     // nicht verwendete Signale für den 1. Schritt und eventuell weitere Schritte
     (*#sxSendBuf.sxSTW1.Jog1          := False;
             #sxSendBuf.sxSTW1.Jog2          := False;
             #sxSendBuf.sxEPosSTW1.MdiTyp    := False;
             #sxSendBuf.sxEPosSTW1.MdiPos    := False;
             #sxSendBuf.sxEPosSTW1.MdiNeg    := False;
             #sxSendBuf.sxEPosSTW1.MdiSetup  := False;
             #sxSendBuf.sxEPosSTW2.SetRefPt  := False;
             #sxSendBuf.sxEPosSTW2.JogInc    := False;
             #sxSendBuf.sxEPosSTW2.RefStDi   := False;
             #sxSendBuf.sxEPosSTW2.RefTyp    := False;
             #sxSendBuf.sxSTW1.RefStart      := False;
             #sxSendBuf.sxEPosSTW1.TrvBit0   := False;
             #sxSendBuf.sxEPosSTW1.TrvBit1   := False;
             #sxSendBuf.sxEPosSTW1.TrvBit2   := False;
             #sxSendBuf.sxEPosSTW1.TrvBit3   := False;
             #sxSendBuf.sxEPosSTW1.TrvBit4   := False;
             #sxSendBuf.sxEPosSTW1.TrvBit5   := False;
             #sxSendBuf.sxEPosSTW1.MdiStart  := False;*)
     #sxSendBuf.STW1.%X8 := False;
     #sxSendBuf.STW1.%X9 := False;
     #sxSendBuf.EPosSTW1.%X8 := False;
     #sxSendBuf.EPosSTW1.%X9 := False;
     #sxSendBuf.EPosSTW1.%X10 := False;
     #sxSendBuf.EPosSTW1.%X14 := False;
     #sxSendBuf.EPosSTW2.%X1 := False;
     #sxSendBuf.EPosSTW2.%X5 := False;
     #sxSendBuf.EPosSTW2.%X9 := False;
     #sxSendBuf.EPosSTW2.%X8 := False;
     #sxSendBuf.STW1.%X11 := False;
     #sxSendBuf.EPosSTW1.%X0 := False;
     #sxSendBuf.EPosSTW1.%X1 := False;
     #sxSendBuf.EPosSTW1.%X2 := False;
     #sxSendBuf.EPosSTW1.%X3 := False;
     #sxSendBuf.EPosSTW1.%X4 := False;
     #sxSendBuf.EPosSTW1.%X5 := False;
     #sxSendBuf.EPosSTW1.%X15 := False;

     // Bei der Auswahl der Verfahrsätze entspricht die Position der Verfahrensatznummer 
     // Verfahrsatznummer aus der Position ermitteln und in die einzelnen Bit's aufteilen
     // Es sind die Verfahrsatznummern 0 - 63 möglich
     IF (DINT_TO_INT(#Position) < 0) OR (DINT_TO_INT(#Position) > 63) THEN
       // Fehler, ungültiger Verfahrsatznummer
       #swStatus := 16#8204;
       #Error := True;
     ELSE
       // Fehler wieder zurücknehmen, wenn er mal ausgelöst wurde
       IF #swStatus = 16#8204 THEN
         #swStatus := 16#7002;
         #Error := False;
       END_IF;

       // Verfahrsatznummer Bit 0 ermitteln
       IF (DINT_TO_WORD(#Position) AND W#16#01) = W#16#01 THEN
         //#sxSendBuf.sxEPosSTW1.TrvBit0 := True;
         #sxSendBuf.EPosSTW1.%X0 := True;
       END_IF;

       // Verfahrsatznummer Bit 1 ermitteln
       IF (DINT_TO_WORD(#Position) AND W#16#02) = W#16#02 THEN
         //#sxSendBuf.sxEPosSTW1.TrvBit1 := True;
         #sxSendBuf.EPosSTW1.%X1 := True;
       END_IF;

       // Verfahrsatznummer Bit 2 ermitteln
       IF (DINT_TO_WORD(#Position) AND W#16#04) = W#16#04 THEN
         //#sxSendBuf.sxEPosSTW1.TrvBit2 := True;
         #sxSendBuf.EPosSTW1.%X2 := True;
       END_IF;

       // Verfahrsatznummer Bit 3 ermitteln
       IF (DINT_TO_WORD(#Position) AND W#16#08) = W#16#08 THEN
         //#sxSendBuf.sxEPosSTW1.TrvBit3 := True;
         #sxSendBuf.EPosSTW1.%X3 := True;
       END_IF;

       // Verfahrsatznummer Bit 4 ermitteln
       IF (DINT_TO_WORD(#Position) AND W#16#10) = W#16#10 THEN
         //#sxSendBuf.sxEPosSTW1.TrvBit4 := True;
         #sxSendBuf.EPosSTW1.%X4 := True;
       END_IF;

       // Verfahrsatznummer Bit 5 ermitteln
       IF (DINT_TO_WORD(#Position) AND W#16#20) = W#16#20 THEN
         //#sxSendBuf.sxEPosSTW1.TrvBit5 := True;
         #sxSendBuf.EPosSTW1.%X5 := True;
       END_IF;

       // Nach dem Einschalten des Antriebes, prüfen ob der Antrieb betriebsbereit, in Operation ohne Fehler und Warnung ist, 
       // dann die Betriebsart MDI / Sollwertvorgabe Start gesetzt werden
       IF #sbOff1 AND #sbReady AND #sbIOp AND NOT #sbFault THEN

         #sxSendBuf.STW1.%X6 := #sbExecute;

         // "Fliegendes Referentieren" aktivieren
         // "Fliegendes Referenzieren" erst nach Einschalten des Antriebes möglich
         IF #sbRefTyp THEN

           // Referenziertyp auf "Fliegendes Referenzieren" einstellen
           //#sxSendBuf.sxEPosSTW2.RefTyp := True;
           #sxSendBuf.EPosSTW2.%X8 := True;

           // Nach der Anwahl des Referenziertyps "Fliegendes Referenzieren", 
           // ein Zyklus später kann das Referenzieren gestartet
           IF (#siRefTypCyc = 0) THEN
             #siRefTypCyc := #siRefTypCyc + 1;
           ELSE
             // Referenzieren starten
             //#sxSendBuf.sxSTW1.RefStart := True;
             #sxSendBuf.STW1.%X11 := True;
           END_IF;
         END_IF;
       END_IF;
     END_IF;

     // Hauptbetriebsart "Tippen" (Jogging)
     // Betriebsart "Tippen positiv" oder "Tippen negativ" angewählt 
   ELSIF #siModePos = 7 AND #sbModePos THEN

     // Antrieb einschalten
     //#sxSendBuf.sxSTW1.Off1 := #sbOff1;
     #sxSendBuf.STW1.%X0 := #sbOff1;

     // nicht verwendete Signale für den 1. Schritt und eventuell weitere Schritte
     (*#sxSendBuf.sxEPosSTW1.MdiStart := False;
             #sxSendBuf.sxEPosSTW2.JogInc   := False;
             #sxSendBuf.sxSTW1.Jog1         := False;
             #sxSendBuf.sxSTW1.Jog2         := False;
             #sxSendBuf.sxEPosSTW2.RefTyp   := False;
             #sxSendBuf.sxSTW1.RefStart     := False;
             #sxSendBuf.sxEPosSTW2.SetRefPt  := False;*)

     #sxSendBuf.EPosSTW1.%X15 := False;
     #sxSendBuf.EPosSTW2.%X5 := False;
     #sxSendBuf.STW1.%X8 := False;
     #sxSendBuf.STW1.%X9 := False;
     #sxSendBuf.EPosSTW2.%X8 := False;
     #sxSendBuf.STW1.%X11 := False;
     #sxSendBuf.EPosSTW2.%X1 := False;

     // Nach dem Einschalten des Antriebes, prüfen ob der Antrieb betriebsbereit, in Operation ohne Fehler und Warnung ist, 
     // dann kann Tippen positiv oder negativ gesetzt werden
     IF #sbOff1 AND #sbReady AND #sbIOp AND NOT #sbFault THEN

       // Tippen positiv
       IF #Jog1 AND NOT #Jog2 THEN
         //#sxSendBuf.sxSTW1.Jog1 := True;
         #sxSendBuf.STW1.%X8 := True;
       END_IF;

       // Tippen negativ
       IF #Jog2 AND NOT #Jog1 THEN
         //#sxSendBuf.sxSTW1.Jog2 := True;
         #sxSendBuf.STW1.%X9 := True;
       END_IF;

       // "Fliegendes Referentieren" aktivieren
       // "Fliegendes Referenzieren" erst nach Einschalten des Antriebes möglich
       IF #sbRefTyp THEN

         // Referenziertyp auf "Fliegendes Referenzieren" einstellen
         //#sxSendBuf.sxEPosSTW2.RefTyp := #FlyRef;
         #sxSendBuf.EPosSTW2.%X8 := #FlyRef;

         // Nach der Anwahl des Referenziertyps "Fliegendes Referenzieren", 
         // ein Zyklus später kann das Referenzieren gestartet
         IF (#siRefTypCyc = 0) THEN
           #siRefTypCyc := #siRefTypCyc + 1;
         ELSE
           // Referenzieren starten
           //#sxSendBuf.sxSTW1.RefStart := True;
           #sxSendBuf.STW1.%X11 := True;
         END_IF;
       END_IF;
     END_IF;

     // Betriebsart "Tippen positiv / Tippen negativ inkrementell" 
   ELSIF #siModePos = 8 AND #sbModePos THEN

     // Antrieb einschalten
     //#sxSendBuf.sxSTW1.OFF1 := #sbOff1;
     #sxSendBuf.STW1.%X0 := #sbOff1;

     // nicht verwendete Signale für den 1. Schritt und eventuell weitere Schritte
     (*#sxSendBuf.sxEPosSTW1.MdiStart := False;
             #sxSendBuf.sxEPosSTW2.JogInc   := False;
             #sxSendBuf.sxSTW1.Jog1         := False;
             #sxSendBuf.sxSTW1.Jog2         := False;
             #sxSendBuf.sxSTW1.RefStart     := False;
             #sxSendBuf.sxEPosSTW2.RefTyp   := False;
             #sxSendBuf.sxEPosSTW2.SetRefPt  := False;*)

     #sxSendBuf.EPosSTW1.%X15 := False;
     #sxSendBuf.EPosSTW2.%X5 := False;
     #sxSendBuf.STW1.%X8 := False;
     #sxSendBuf.STW1.%X9 := False;
     #sxSendBuf.STW1.%X11 := False;
     #sxSendBuf.EPosSTW2.%X8 := False;
     #sxSendBuf.EPosSTW2.%X1 := False;

     // Nach dem Einschalten des Antriebes, ein Paar Zyklen warten bevor Tippen negativ gesetzt werden kann
     // Nach dem Einschalten des Antriebes, prüfen ob der Antrieb betriebsbereit, in Operation ohne Fehler und Warnung ist, 
     // dann kann Tippen positiv oder negativ gesetzt werden
     IF #sbOff1 AND #sbReady AND #sbIOp AND NOT #sbFault THEN

       // Tippen inkrementell einstellen
       //#sxSendBuf.sxEPosSTW2.JogInc := True;
       #sxSendBuf.EPosSTW2.%X5 := True;

       #sbJogInc := True;

       // Nach dem Einstellen des Antriebes, ein Paar Zyklen warten bevor Tippen negativ oder Tippen positiv gesetz werden kann
       IF #sbJogInc AND (#siJogIncCyc = 0) THEN
         #siJogIncCyc := #siJogIncCyc + 1;
       ELSE

         // Tippen positiv oder negativ inkrementell zulassen
         IF #Jog1 XOR #Jog2 THEN

           //#sxSendBuf.sxSTW1.Jog1 := #Jog1;
           //#sxSendBuf.sxSTW1.Jog2 := #Jog2;
           #sxSendBuf.STW1.%X8 := #Jog1;
           #sxSendBuf.STW1.%X9 := #Jog2;
         END_IF;
       END_IF;

       // "Fliegendes Referentieren" aktivieren
       // "Fliegendes Referenzieren" erst nach Einschalten des Antriebes möglich
       IF #sbRefTyp THEN

         // Referenziertyp auf "Fliegendes Referenzieren" einstellen
         //#sxSendBuf.sxEPosSTW2.RefTyp := True;
         #sxSendBuf.EPosSTW2.%X8 := True;

         // Nach der Anwahl des Referenziertyps "Fliegendes Referenzieren", 
         // ein Zyklus später kann das Referenzieren gestartet
         IF (#siRefTypCyc = 0) THEN
           #siRefTypCyc := #siRefTypCyc + 1;
         ELSE
           // Referenzieren starten
           //#sxSendBuf.sxSTW1.RefStart := True;
           #sxSendBuf.STW1.%X11 := True;
         END_IF;
       END_IF;
     END_IF;
   ELSE
     // Werte wieder zurücknehmen
     (*#sxSendBuf.sxSTW1.Off1          := #Off1;
             #sxSendBuf.sxSTW1.RejTrvTsk     := False;
             #sxSendBuf.sxSTW1.TrvStart      := False;
             #sxSendBuf.sxEPosSTW1.MdiStart  := False;
             #sxSendBuf.sxSTW1.Jog1          := False;
             #sxSendBuf.sxSTW1.Jog2          := False;
             #sxSendBuf.sxEPosSTW1.MdiTyp    := False;
             #sxSendBuf.sxEPosSTW1.MdiPos    := False;
             #sxSendBuf.sxEPosSTW1.MdiNeg    := False;
             #sxSendBuf.sxEPosSTW1.MdiTrTyp  := False;
             #sxSendBuf.sxEPosSTW1.MdiSetup  := False;
             #sxSendBuf.sxEPosSTW2.SetRefPt  := False;
             #sxSendBuf.sxEPosSTW2.RefTyp    := False;
             #sxSendBuf.sxEPosSTW2.RefStDi   := False;
             #sxSendBuf.sxEPosSTW2.JogInc    := False;
             #sxSendBuf.sxSTW1.RefStart      := False;*)

     #sxSendBuf.STW1.%X0 := #EnableAxis;
     #sxSendBuf.STW1.%X4 := False;
     #sxSendBuf.STW1.%X6 := False;
     #sxSendBuf.EPosSTW1.%X15 := False;
     #sxSendBuf.STW1.%X8 := False;
     #sxSendBuf.STW1.%X9 := False;
     #sxSendBuf.EPosSTW1.%X8 := False;
     #sxSendBuf.EPosSTW1.%X9 := False;
     #sxSendBuf.EPosSTW1.%X10 := False;
     #sxSendBuf.EPosSTW1.%X12 := False;
     #sxSendBuf.EPosSTW1.%X14 := False;
     #sxSendBuf.EPosSTW2.%X1 := False;
     #sxSendBuf.EPosSTW2.%X8 := False;
     #sxSendBuf.EPosSTW2.%X9 := False;
     #sxSendBuf.EPosSTW2.%X5 := False;
     #sxSendBuf.STW1.%X11 := False;
   END_IF; // Hauptbetriebsart "Verfahrsätze" (Traversing Blocks)

   //Den Eingang ConfigEPos auf die einzelnen Bits im Telegramm verschalten
   #sxSendBuf.STW1.%X1 := #ConfigEPos.%X0;
   #sxSendBuf.STW1.%X2 := #ConfigEPos.%X1;
   #sxSendBuf.EPosSTW2.%X14 := #ConfigEPos.%X2;
   #sxSendBuf.EPosSTW2.%X15 := #ConfigEPos.%X3;
   #sxSendBuf.EPosSTW2.%X11 := #ConfigEPos.%X4;
   #sxSendBuf.EPosSTW2.%X10 := #ConfigEPos.%X5;
   #sxSendBuf.EPosSTW2.%X2 := #ConfigEPos.%X6;
   #sxSendBuf.STW1.%X13 := #ConfigEPos.%X7;
   #sxSendBuf.EPosSTW1.%X12 := #ConfigEPos.%X8;
   #sxSendBuf.STW2.%X0 := #ConfigEPos.%X9;
   #sxSendBuf.STW2.%X1 := #ConfigEPos.%X10;
   #sxSendBuf.STW2.%X2 := #ConfigEPos.%X11;
   #sxSendBuf.STW2.%X3 := #ConfigEPos.%X12;
   #sxSendBuf.STW2.%X4 := #ConfigEPos.%X13;
   #sxSendBuf.STW2.%X7 := #ConfigEPos.%X14;
   #sxSendBuf.STW1.%X12 := #ConfigEPos.%X15;
   #sxSendBuf.STW1.%X14 := #ConfigEPos.%X16;
   #sxSendBuf.STW1.%X15 := #ConfigEPos.%X17;
   #sxSendBuf.EPosSTW1.%X6 := #ConfigEPos.%X18;
   #sxSendBuf.EPosSTW1.%X7 := #ConfigEPos.%X19;
   #sxSendBuf.EPosSTW1.%X11 := #ConfigEPos.%X20;
   #sxSendBuf.EPosSTW1.%X13 := #ConfigEPos.%X21;
   #sxSendBuf.EPosSTW2.%X3 := #ConfigEPos.%X22;
   #sxSendBuf.EPosSTW2.%X4 := #ConfigEPos.%X23;
   #sxSendBuf.EPosSTW2.%X6 := #ConfigEPos.%X24;
   #sxSendBuf.EPosSTW2.%X7 := #ConfigEPos.%X25;
   #sxSendBuf.EPosSTW2.%X12 := #ConfigEPos.%X26;
   #sxSendBuf.EPosSTW2.%X13 := #ConfigEPos.%X27;
   #sxSendBuf.STW2.%X5 := #ConfigEPos.%X28;
   #sxSendBuf.STW2.%X6 := #ConfigEPos.%X29;
   #sxSendBuf.STW2.%X8 := #ConfigEPos.%X30;
   #sxSendBuf.STW2.%X9 := #ConfigEPos.%X31;


   #swSendBuf[0] := #sxSendBuf.STW1;
   #swSendBuf[1] := #sxSendBuf.EPosSTW1;
   #swSendBuf[2] := #sxSendBuf.EPosSTW2;
   #swSendBuf[3] := #sxSendBuf.STW2;
   #swSendBuf[4] := #sxSendBuf.OverrideV;
   #swSendBuf[5] := #sxSendBuf.Position.%W1;
   #swSendBuf[6] := #sxSendBuf.Position.%W0;
   #swSendBuf[7] := #sxSendBuf.Velocity.%W1;
   #swSendBuf[8] := #sxSendBuf.Velocity.%W0;
   #swSendBuf[9] := #sxSendBuf.OverrideA;
   #swSendBuf[10] := #sxSendBuf.OverrideD;
   #swSendBuf[11] := #sxSendBuf.Reserve;

   //Prozessdaten zur Signalbaugruppe schreiben
   #piRetSFC := DPWR_DAT(LADDR := #HWIDSTW,
                         RECORD := #swSendBuf);

   // Fehler der Rückmeldung ausgeben
   #DiagID := INT_TO_WORD(#piRetSFC);

   //kein Fehler beim Schreiben
   IF #piRetSFC = 0 THEN

     // Fehler wieder zurück nehmen
     IF (#swStatus = 16#8601) THEN
       #swStatus := 16#7002;
       #Error := False;
     END_IF;

     //Prozessdaten von der Signalbaugruppe lesen
     #piRetSFC := DPRD_DAT(LADDR := #HWIDZSW,
                           RECORD => #swRecvBuf);

     // Fehlermeldung der Rückmeldung ausgeben
     #DiagID := INT_TO_WORD(#piRetSFC);

     //Fehler beim Lesen (Profibus-Kommunikation unterbrochen)
     IF #piRetSFC <> 0 THEN

       // Fehler
       #Error := TRUE;
       #swStatus := 16#8600;

       // Zustandsworte löschen
       #sxRecvBuf.ZSW1 := W#16#0;
       #sxRecvBuf.EPosZSW1 := W#16#0;
       #sxRecvBuf.EPosZSW2 := W#16#0;
       #sxRecvBuf.ZSW2 := W#16#0;
       #sxRecvBuf.NotUsed := W#16#00;
       #sxRecvBuf.Position := DW#16#00;
       #sxRecvBuf.Velocity := DW#16#00;
       #sxRecvBuf.ErrNr := W#16#00;
       #sxRecvBuf.WarnNr := W#16#00;
       #sxRecvBuf.Reserve := W#16#00;

       // Werte auslesen
     ELSE

       // Fehler wieder zurück nehmen
       IF (#swStatus = 16#8600) THEN
         #swStatus := 16#7002;
         #Error := False;
       END_IF;

       #sxRecvBuf.ZSW1 := #swRecvBuf[0];
       #sxRecvBuf.EPosZSW1 := #swRecvBuf[1];
       #sxRecvBuf.EPosZSW2 := #swRecvBuf[2];
       #sxRecvBuf.ZSW2 := #swRecvBuf[3];
       #sxRecvBuf.NotUsed := #swRecvBuf[4];
       #sxRecvBuf.Position.%W1 := #swRecvBuf[5];
       #sxRecvBuf.Position.%W0 := #swRecvBuf[6];
       #sxRecvBuf.Velocity.%W1 := #swRecvBuf[7];
       #sxRecvBuf.Velocity.%W0 := #swRecvBuf[8];
       #sxRecvBuf.ErrNr := #swRecvBuf[9];
       #sxRecvBuf.WarnNr := #swRecvBuf[10];
       #sxRecvBuf.Reserve := #swRecvBuf[11];

       // ZSW1 aufbereiten
       //#Busy := #sxRecvBuf.sxZSW1.IOp;
       #sbBusy := #sxRecvBuf.ZSW1.%X2;

       // Fehler auswerten
       IF #sxRecvBuf.ZSW1.%X3 THEN
         #swStatus := 16#8401;
         #Error := True;
       ELSIF #sxRecvBuf.ZSW1.%X6 THEN
         #swStatus := 16#8402;
         #Error := True;
       ELSE
         // Fehler wieder zurück nehmen
         IF (#swStatus = 16#8401) OR (#swStatus = 16#8402) THEN
           #swStatus := 16#7002;
           #Error := False;
         END_IF;
       END_IF;

       // EPOS_ZSW1            
       // EPOS-Wort-1 BIT 00 --> 1 = Active traversing block bit 0
       //IF #sxRecvBuf.sxEPosZSW1.ActTrvBit0 THEN
       IF #sxRecvBuf.EPosZSW1.%X0 THEN
         #swEPosZSW1 := #swEPosZSW1 OR W#16#01;
       ELSE
         #swEPosZSW1 := #swEPosZSW1 AND W#16#FFFE;
       END_IF;

       // EPOS-Wort-1 Bit 01 --> 1 = Active traversing block bit 1
       //IF #sxRecvBuf.sxEPosZSW1.ActTrvBit1 THEN
       IF #sxRecvBuf.EPosZSW1.%X1 THEN
         #swEPosZSW1 := #swEPosZSW1 OR W#16#02;
       ELSE
         #swEPosZSW1 := #swEPosZSW1 AND W#16#FFFD;
       END_IF;

       // EPOS-Wort-1 Bit 02 --> 1 = Active traversing block bit 2
       //IF #sxRecvBuf.sxEPosZSW1.ActTrvBit2 THEN
       IF #sxRecvBuf.EPosZSW1.%X2 THEN
         #swEPosZSW1 := #swEPosZSW1 OR W#16#04;
       ELSE
         #swEPosZSW1 := #swEPosZSW1 AND W#16#FFFB;
       END_IF;

       // EPOS-Wort-1 Bit 03 --> 1 = Active traversing block bit 3
       //IF #sxRecvBuf.sxEPosZSW1.ActTrvBit3 THEN
       IF #sxRecvBuf.EPosZSW1.%X3 THEN
         #swEPosZSW1 := #swEPosZSW1 OR W#16#08;
       ELSE
         #swEPosZSW1 := #swEPosZSW1 AND W#16#FFF7;
       END_IF;(*

   *)

       // EPOS-Wort-1 Bit 04 --> 1 = Active traversing block bit 4 
       //IF #sxRecvBuf.sxEPosZSW1.ActTrvBit4 THEN
       IF #sxRecvBuf.EPosZSW1.%X4 THEN
         #swEPosZSW1 := #swEPosZSW1 OR W#16#10;
       ELSE
         #swEPosZSW1 := #swEPosZSW1 AND W#16#FFEF;
       END_IF;

       // EPOS-Wort-1 Bit 05 --> 1 = Active traversing block bit 5
       //IF #sxRecvBuf.sxEPosZSW1.ActTrvBit5 THEN
       IF #sxRecvBuf.EPosZSW1.%X5 THEN
         #swEPosZSW1 := #swEPosZSW1 OR W#16#20;
       ELSE
         #swEPosZSW1 := #swEPosZSW1 AND W#16#FFDF;
       END_IF;

       // EPOS-Wort-1 Bit 08 --> 1 = STOP cam minus active
       //IF #sxRecvBuf.sxEPosZSW1.StpCamMinAct THEN
       IF #sxRecvBuf.EPosZSW1.%X8 THEN
         #swEPosZSW1 := #swEPosZSW1 OR W#16#100;
       ELSE
         #swEPosZSW1 := #swEPosZSW1 AND W#16#FEFF;
       END_IF;

       // EPOS-Wort-1 Bit 09 --> 1 = STOP cam plus active
       //IF #sxRecvBuf.sxEPosZSW1.StpCamPlsAct THEN
       IF #sxRecvBuf.EPosZSW1.%X9 THEN
         #swEPosZSW1 := #swEPosZSW1 OR W#16#200;
       ELSE
         #swEPosZSW1 := #swEPosZSW1 AND W#16#FDFF;
       END_IF;

       // EPOS-Wort-1 Bit 10 --> 1 = Jogging active
       //IF #sxRecvBuf.sxEPosZSW1.JogAct THEN
       IF #sxRecvBuf.EPosZSW1.%X10 THEN
         #swEPosZSW1 := #swEPosZSW1 OR W#16#400;
       ELSE
         #swEPosZSW1 := #swEPosZSW1 AND W#16#FBFF;
       END_IF;

       // EPOS-Wort-1 Bit 11 --> 1 = Reference point approach active
       //IF #sxRecvBuf.sxEPosZSW1.RefAct THEN
       IF #sxRecvBuf.EPosZSW1.%X11 THEN
         #swEPosZSW1 := #swEPosZSW1 OR W#16#800;
       ELSE
         #swEPosZSW1 := #swEPosZSW1 AND W#16#F7FF;
       END_IF;

       // Anstossen des fliegenden Referenzieren prüfen, wenn die Rückmeldung fehlt dann wiederholen
       //IF NOT #sxRecvBuf.sxEPosZSW1.FlyRefAct AND #sbRefTyp AND #sxSendBuf.sxSTW1.RefStart THEN
       IF NOT #sxRecvBuf.EPosZSW1.%X12 AND #sbRefTyp AND #sxSendBuf.STW1.%X11 THEN

         // Wiederholung anstossen 
         IF #siRefActRetry < #siRetryMax THEN
           #siRefActRetry := #siRefActRetry + 1;

           // Referenzieren starten wieder wegnehmen
           //#sxSendBuf.sxSTW1.RefStart := False;
           #sxSendBuf.STW1.%X11 := False;
         ELSE

           // Fehlermeldung
           #swStatus := 16#8403;
           #Error := True;
         END_IF;
       ELSE

         // Fehler wieder zurücknehmen, wenn er mal ausgelöst wurde
         IF #swStatus = 16#8403 THEN
           #swStatus := 16#7002;
           #Error := False;
         END_IF;
         // Zähler zurücksetzen bei Rückmeldung fliegendes Referenzieren jetzt aktiviert oder bei Abwahl der Funktion
         IF (#sxRecvBuf.EPosZSW1.%X12 AND #sbRefTyp AND #sxSendBuf.STW1.%X11) OR NOT #FlyRef THEN
           #siRefActRetry := 0;
         END_IF;
       END_IF;

       // EPOS-Wort-1 Bit 12 --> 1 = Flying referencing active
       //IF #sxRecvBuf.sxEPosZSW1.FlyRefAct THEN
       IF #sxRecvBuf.EPosZSW1.%X12 THEN
         #swEPosZSW1 := #swEPosZSW1 OR W#16#1000;
       ELSE
         #swEPosZSW1 := #swEPosZSW1 AND W#16#EFFF;
       END_IF;

       // EPOS-Wort-1 Bit 13 --> 1 = Traversing block active
       //IF #sxRecvBuf.sxEPosZSW1.TrvBlAct THEN
       IF #sxRecvBuf.EPosZSW1.%X13 THEN
         #swEPosZSW1 := #swEPosZSW1 OR W#16#2000;
       ELSE
         #swEPosZSW1 := #swEPosZSW1 AND W#16#DFFF;
       END_IF;

       // EPOS-Wort-1 Bit 14 --> 1 = MDI setup active
       //IF #sxRecvBuf.sxEPosZSW1.MdiStupAct THEN
       IF #sxRecvBuf.EPosZSW1.%X14 THEN
         #swEPosZSW1 := #swEPosZSW1 OR W#16#4000;
       ELSE
         #swEPosZSW1 := #swEPosZSW1 AND W#16#BFFF;
       END_IF;

       // EPOS-Wort-1 Bit 15 --> 1 = MDI positing active
       //IF #sxRecvBuf.sxEPosZSW1.MdiPosAct THEN
       IF #sxRecvBuf.EPosZSW1.%X15 THEN
         #swEPosZSW1 := #swEPosZSW1 OR W#16#8000;
       ELSE
         #swEPosZSW1 := #swEPosZSW1 AND W#16#7FFF;
       END_IF;

       // EPOS_ZSW2 
       // EPOS-Wort-2 Bit 00 --> 1 = Tracking mode active
       //IF #sxRecvBuf.sxEPosZSW2.TrkModeAct THEN
       IF #sxRecvBuf.EPosZSW2.%X0 THEN
         #swEPosZSW2 := #swEPosZSW2 OR W#16#01;
       ELSE
         #swEPosZSW2 := #swEPosZSW2 AND W#16#FFFE;
       END_IF;

       // EPOS-Wort-2 Bit 01 --> 1 = Velocity limit active
       //IF #sxRecvBuf.sxEPosZSW2.VeloLimAct THEN
       IF #sxRecvBuf.EPosZSW2.%X1 THEN
         #swEPosZSW2 := #swEPosZSW2 OR W#16#02;
       ELSE
         #swEPosZSW2 := #swEPosZSW2 AND W#16#FFFD;
       END_IF;

       // EPOS-Wort-2 Bit 02 --> 1 = Setpoint static
       //IF #sxRecvBuf.sxEPosZSW2.SetPStat THEN
       IF #sxRecvBuf.EPosZSW2.%X2 THEN
         #swEPosZSW2 := #swEPosZSW2 OR W#16#04;
       ELSE
         #swEPosZSW2 := #swEPosZSW2 AND W#16#FFFB;
       END_IF;

       // EPOS-Wort-2 Bit 03 --> 1 = Printmark outside outer window
       //IF #sxRecvBuf.sxEPosZSW2.PrnMrkOut THEN
       IF #sxRecvBuf.EPosZSW2.%X3 THEN
         #swEPosZSW2 := #swEPosZSW2 OR W#16#08;
       ELSE
         #swEPosZSW2 := #swEPosZSW2 AND W#16#FFF7;
       END_IF;

       // EPOS-Wort-2 Bit 04 --> 1 = Axis forwards
       //IF #sxRecvBuf.sxEPosZSW2.FWD THEN
       IF #sxRecvBuf.EPosZSW2.%X4 THEN
         #swEPosZSW2 := #swEPosZSW2 OR W#16#10;
       ELSE
         #swEPosZSW2 := #swEPosZSW2 AND W#16#FFEF;
       END_IF;

       // EPOS-Wort-2 Bit 05 --> 1 = Axis backwards
       //IF #sxRecvBuf.sxEPosZSW2.BWD THEN
       IF #sxRecvBuf.EPosZSW2.%X5 THEN
         #swEPosZSW2 := #swEPosZSW2 OR W#16#20;
       ELSE
         #swEPosZSW2 := #swEPosZSW2 AND W#16#FFDF;
       END_IF;

       // EPOS-Wort-2 Bit 06 --> 1 = Software limit switch minus active
       //IF #sxRecvBuf.sxEPosZSW2.SftSwMinAct THEN
       IF #sxRecvBuf.EPosZSW2.%X6 THEN
         #swEPosZSW2 := #swEPosZSW2 OR W#16#40;
       ELSE
         #swEPosZSW2 := #swEPosZSW2 AND W#16#FFBF;
       END_IF;

       // EPOS-Wort-2 Bit 07 --> 1 = Software limit switch plus active
       //IF #sxRecvBuf.sxEPosZSW2.SftSwPlsAct THEN
       IF #sxRecvBuf.EPosZSW2.%X7 THEN
         #swEPosZSW2 := #swEPosZSW2 OR W#16#80;
       ELSE
         #swEPosZSW2 := #swEPosZSW2 AND W#16#FF7F;
       END_IF;

       // EPOS-Wort-2 Bit 08 --> 1 = Position actual value <= cam position 1
       //IF #sxRecvBuf.sxEPosZSW2.PosSmCam1 THEN
       IF #sxRecvBuf.EPosZSW2.%X8 THEN
         #swEPosZSW2 := #swEPosZSW2 OR W#16#100;
       ELSE
         #swEPosZSW2 := #swEPosZSW2 AND W#16#FEFF;
       END_IF;

       // EPOS-Wort-2 Bit 09 --> 1 = Position actual value <= cam position 2
       //IF #sxRecvBuf.sxEPosZSW2.PosSmCam2 THEN
       IF #sxRecvBuf.EPosZSW2.%X9 THEN
         #swEPosZSW2 := #swEPosZSW2 OR W#16#200;
       ELSE
         #swEPosZSW2 := #swEPosZSW2 AND W#16#FDFF;
       END_IF;

       // EPOS-Wort-2 Bit 10 --> 1 = Direct output 1 via traversing block
       //IF #sxRecvBuf.sxEPosZSW2.TrvOut1 THEN
       IF #sxRecvBuf.EPosZSW2.%X10 THEN
         #swEPosZSW2 := #swEPosZSW2 OR W#16#400;
       ELSE
         #swEPosZSW2 := #swEPosZSW2 AND W#16#FBFF;
       END_IF;

       // EPOS-Wort-2 Bit 11 --> 1 = Direct output 2 via traversing block
       //IF #sxRecvBuf.sxEPosZSW2.TrvOut2 THEN
       IF #sxRecvBuf.EPosZSW2.%X11 THEN
         #swEPosZSW2 := #swEPosZSW2 OR W#16#800;
       ELSE
         #swEPosZSW2 := #swEPosZSW2 AND W#16#F7FF;
       END_IF;

       // EPOS-Wort-2 Bit 12 --> 1 = Fixed STOP reached
       //IF #sxRecvBuf.sxEPosZSW2.FxStpRd THEN
       IF #sxRecvBuf.EPosZSW2.%X12 THEN
         #swEPosZSW2 := #swEPosZSW2 OR W#16#1000;
       ELSE
         #swEPosZSW2 := #swEPosZSW2 AND W#16#EFFF;
       END_IF;

       // EPOS-Wort-2 Bit 13 --> 1 = Fixed STOP clamping torque reached
       //IF #sxRecvBuf.sxEPosZSW2.FxStpTrRd THEN
       IF #sxRecvBuf.EPosZSW2.%X13 THEN
         #swEPosZSW2 := #swEPosZSW2 OR W#16#2000;
       ELSE
         #swEPosZSW2 := #swEPosZSW2 AND W#16#DFFF;
       END_IF;

       // EPOS-Wort-2 Bit 14 --> 1 = Traversing fixed STOP active
       //IF #sxRecvBuf.sxEPosZSW2.TrvFxStpAct THEN
       IF #sxRecvBuf.EPosZSW2.%X14 THEN
         #swEPosZSW2 := #swEPosZSW2 OR W#16#4000;
       ELSE
         #swEPosZSW2 := #swEPosZSW2 AND W#16#BFFF;
       END_IF;

       // EPOS-Wort-2 Bit 15 --> 1 = Traversing command active
       //IF #sxRecvBuf.sxEPosZSW2.CmdAct THEN
       IF #sxRecvBuf.EPosZSW2.%X15 THEN
         #swEPosZSW2 := #swEPosZSW2 OR W#16#8000;
       ELSE
         #swEPosZSW2 := #swEPosZSW2 AND W#16#7FFF;
       END_IF;

       #sbReady := #sxRecvBuf.ZSW1.%X1;

       #AxisEnabled := #sxRecvBuf.ZSW1.%X2;
       #sbIOp := #sxRecvBuf.ZSW1.%X2;

       #AxisError := #sxRecvBuf.ZSW1.%X3;
       #sbFault := #sxRecvBuf.ZSW1.%X3;

       #AxisWarn := #sxRecvBuf.ZSW1.%X7;
       #sbAlarm := #sxRecvBuf.ZSW1.%X7;

       #AxisPosOk := #sxRecvBuf.ZSW1.%X10;
       #AxisRef := #sxRecvBuf.ZSW1.%X11;
       #AxisSpFixed := #sxRecvBuf.ZSW1.%X13;

       #sbAccel := #sxRecvBuf.ZSW1.%X14;
       #sbDecel := #sxRecvBuf.ZSW1.%X15;

       #ActVelocity := DWORD_TO_DINT(#sxRecvBuf.Velocity);
       #ActPosition := DWORD_TO_DINT(#sxRecvBuf.Position);
       #ActMode := #ModePos;
       #ActWarn := #sxRecvBuf.WarnNr;
       #ActFault := #sxRecvBuf.ErrNr;

       #Lockout := #sxRecvBuf.ZSW1.%X6;
     END_IF;
   ELSE

     // Fehler
     #Error := TRUE;
     #swStatus := 16#8601;

   END_IF;

   // Initialisierung von Ausg㭧en
   #Status := #swStatus;
   #EPosZSW1 := #swEPosZSW1;
   #EPosZSW2 := #swEPosZSW2;
END_FUNCTION_BLOCK

// folder: General

FUNCTION_BLOCK "InOut"   // FB1, LAD
{ S7_Optimized_Access := 'TRUE' }
VERSION : 0.1
   VAR
      BaseDrive_LAD_Instance : "BaseDrive_LAD";
      CiftEl_Instance : "CiftEl";
   END_VAR
   VAR_TEMP
      bHmiServoStopButton : Bool;
      bDriveEnable : Bool;
   END_VAR
BEGIN

REGION Network 1: Cift El
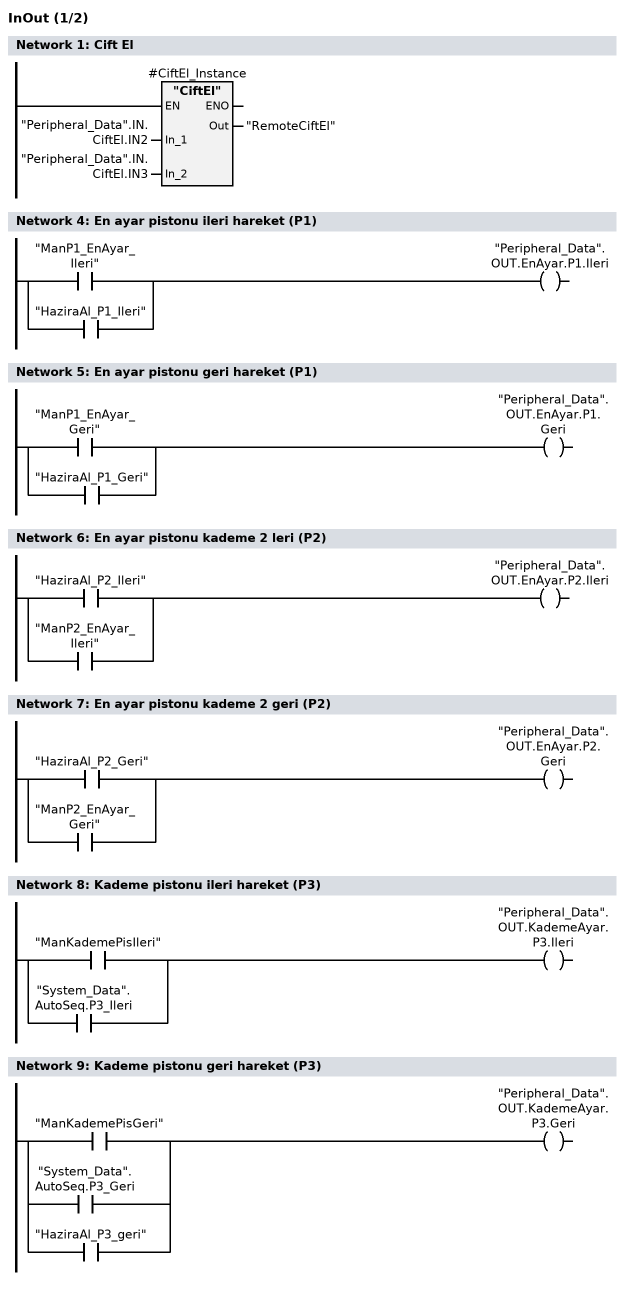
   RUNG wire#powerrail
      #CiftEl_Instance(In_1 := "Peripheral_Data".IN.CiftEl.IN2, In_2 := "Peripheral_Data".IN.CiftEl.IN3, Out => "RemoteCiftEl")
   END_RUNG
   // the same network as SCL:
   #CiftEl_Instance(In_1 := "Peripheral_Data".IN.CiftEl.IN2,   // "CiftEl"
                    In_2 := "Peripheral_Data".IN.CiftEl.IN3,
                    Out => "RemoteCiftEl");
END_REGION

REGION Network 2 (SCL): Servo veri yonetimi

   //********************************************//
   //******* Servo Poizsyona git işlemleri*******//
   "System_Data".CmdDrive.GoPos :=
   "ManServoGoPos" OR "System_Data".AutoSeq.GoPos
   OR "System_Data".AutoSeq.GoPos2 OR "HaziraAl_ServoGoPos"
   OR "ManServoGoHome" OR "ManServoGoPos2";

   //**********************************************//
   //********* Manuel jog kontrolleri*************//
   "System_Data".CmdDrive.Jog1 := "ManServoJog1";
   "System_Data".CmdDrive.Jog2 := "ManServoJog2";

   "System_Data".CmdDrive.SetReference := "System_Data".SystemMode.Man AND "HMI_Data".ServoButton.btnRefNokBelirle;
   "System_Data".CmdDrive.AckError := "System_Data".SystemMode.Man AND "HMI_Data".ServoButton.btnHataReset;
   //"System_Data".CmdDrive.Position := "Receipt".CurrentModel.Boy_C;

   //************************************************//
   //*********Servo hız bilgisi**********************//
   //

   "System_Data".CmdDrive.Velocity := 30.0;
   "System_Data".CmdDrive.Override := "HMI_Data".ServoData.txtJogOverride;  // jog hızı

   // IF "System_Data".SystemMode.Auto THEN
   //     //"System_Data".CmdDrive.Velocity := "HMI_Data".ServoData.txtVelocity;  //otomatik sekans hızı
   //     "System_Data".CmdDrive.Velocity := INT_TO_REAL("HMI_Data".ServoData.txtJogOverride);
   //     "System_Data".CmdDrive.Override := 100; 
   // ELSIF "System_Data".SystemMode.Man THEN
   //     "System_Data".CmdDrive.Velocity := INT_TO_REAL( "HMI_Data".ServoData.txtJogOverride );
   //     "System_Data".CmdDrive.Override := "HMI_Data".ServoData.txtJogOverride;  // jog hızı
   // END_IF;

   //***********************************************//
   //********** Home Konumu ************************//
   "System_Data".CmdDrive.HomePosition := 1560.0;
END_REGION

REGION Network 3 (SCL): Drive blogu
   // Hmi servo ekranı stop butonu sadece manuel modda çalışacak
   #bHmiServoStopButton := "HMI_Data".ServoButton.btnStop AND "System_Data".SystemMode.Man;
   #bDriveEnable := "System_Data".AutoSeq.StartedInfo
                   OR "HaziraAl_ServoGoPos"
                   OR "ManServoGoPos"
                   OR "ManServoGoPos2"
                   OR "ManServoGoHome"
                   OR "System_Data".CmdDrive.SetReference;

   #BaseDrive_LAD_Instance(Emergency := "Peripheral_Data".IN.Acil_Stop,
                           //Enable := #bDriveEnable,
                           Enable := "Peripheral_Data".IN.Acil_Stop AND NOT "HMI_Data".btnStop AND NOT #bHmiServoStopButton,
                           GoPos:="System_Data".CmdDrive.GoPos,
                           //GoHome:="System_Data".CmdDrive.GoHome,
                           SetReference:="System_Data".CmdDrive.SetReference,
                           Jog1:="System_Data".CmdDrive.Jog1,
                           Jog2:="System_Data".CmdDrive.Jog2,
                           Position:="System_Data".CmdDrive.Position,
                           Velocity:="System_Data".CmdDrive.Velocity,
                           Override:="System_Data".CmdDrive.Override,
                           AckError:="System_Data".CmdDrive.AckError,
                           HWDSTW:=280,
                           HWDZSW:=280,
                           Pos_Done=>"System_Data".CmdDrive.Pos_Done,
                           Busy=>"System_Data".CmdDrive.Busy,
                           Error=>"System_Data".CmdDrive.Error,
                           AxisError => "System_Data".CmdDrive.AxisError,
                           ErrorId=>"System_Data".CmdDrive.ErrorId,
                           ReferencedAxis=>"System_Data".CmdDrive.ReferencedAxis,
                           Message=>"System_Data".CmdDrive.Message,
                           ActPosition=>"System_Data".CmdDrive.ActPosition,
                           Alarm=>"System_Data".CmdDrive.Alarm,
                           //IsHomePosTol => "System_Data".CmdDrive.IsHomePosTol,
                           IsPosTol => "System_Data".CmdDrive.IsPosTol,
                           Standstill => "MemDrive_Standsill");

   "HMI_Data".ServoData.txtActPozisyon := "System_Data".CmdDrive.ActPosition;
END_REGION

REGION Network 4: En ayar pistonu ileri hareket (P1)
   RUNG wire#powerrail
      Contact( "ManP1_EnAyar_Ileri" )
      wire#w1
      Coil( "Peripheral_Data".OUT.EnAyar.P1.Ileri )
   END_RUNG
   RUNG wire#powerrail
      Contact( "HaziraAl_P1_Ileri" )
   END_RUNG wire#w1
   // the same network as SCL:
   "Peripheral_Data".OUT.EnAyar.P1.Ileri := "ManP1_EnAyar_Ileri" OR "HaziraAl_P1_Ileri";
END_REGION

REGION Network 5: En ayar pistonu geri hareket (P1)
   RUNG wire#powerrail
      Contact( "ManP1_EnAyar_Geri" )
      wire#w1
      Coil( "Peripheral_Data".OUT.EnAyar.P1.Geri )
   END_RUNG
   RUNG wire#powerrail
      Contact( "HaziraAl_P1_Geri" )
   END_RUNG wire#w1
   // the same network as SCL:
   "Peripheral_Data".OUT.EnAyar.P1.Geri := "ManP1_EnAyar_Geri" OR "HaziraAl_P1_Geri";
END_REGION

REGION Network 6: En ayar pistonu kademe 2 leri (P2)
   RUNG wire#powerrail
      Contact( "HaziraAl_P2_Ileri" )
      wire#w1
      Coil( "Peripheral_Data".OUT.EnAyar.P2.Ileri )
   END_RUNG
   RUNG wire#powerrail
      Contact( "ManP2_EnAyar_Ileri" )
   END_RUNG wire#w1
   // the same network as SCL:
   "Peripheral_Data".OUT.EnAyar.P2.Ileri := "HaziraAl_P2_Ileri" OR "ManP2_EnAyar_Ileri";
END_REGION

REGION Network 7: En ayar pistonu kademe 2 geri (P2)
   RUNG wire#powerrail
      Contact( "HaziraAl_P2_Geri" )
      wire#w1
      Coil( "Peripheral_Data".OUT.EnAyar.P2.Geri )
   END_RUNG
   RUNG wire#powerrail
      Contact( "ManP2_EnAyar_Geri" )
   END_RUNG wire#w1
   // the same network as SCL:
   "Peripheral_Data".OUT.EnAyar.P2.Geri := "HaziraAl_P2_Geri" OR "ManP2_EnAyar_Geri";
END_REGION

REGION Network 8: Kademe pistonu ileri hareket (P3)
   RUNG wire#powerrail
      Contact( "ManKademePisIleri" )
      wire#w1
      Coil( "Peripheral_Data".OUT.KademeAyar.P3.Ileri )
   END_RUNG
   RUNG wire#powerrail
      Contact( "System_Data".AutoSeq.P3_Ileri )
   END_RUNG wire#w1
   // the same network as SCL:
   "Peripheral_Data".OUT.KademeAyar.P3.Ileri := "ManKademePisIleri" OR "System_Data".AutoSeq.P3_Ileri;
END_REGION

REGION Network 9: Kademe pistonu geri hareket (P3)
   RUNG wire#powerrail
      Contact( "ManKademePisGeri" )
      wire#w1
      Coil( "Peripheral_Data".OUT.KademeAyar.P3.Geri )
   END_RUNG
   RUNG wire#powerrail
      Contact( "System_Data".AutoSeq.P3_Geri )
   END_RUNG wire#w1
   RUNG wire#powerrail
      Contact( "HaziraAl_P3_geri" )
   END_RUNG wire#w1
   // the same network as SCL:
   "Peripheral_Data".OUT.KademeAyar.P3.Geri := "ManKademePisGeri" OR "System_Data".AutoSeq.P3_Geri OR "HaziraAl_P3_geri";
END_REGION

REGION Network 10: Kenetleme pistonu ileri hareket (P4/P4B)
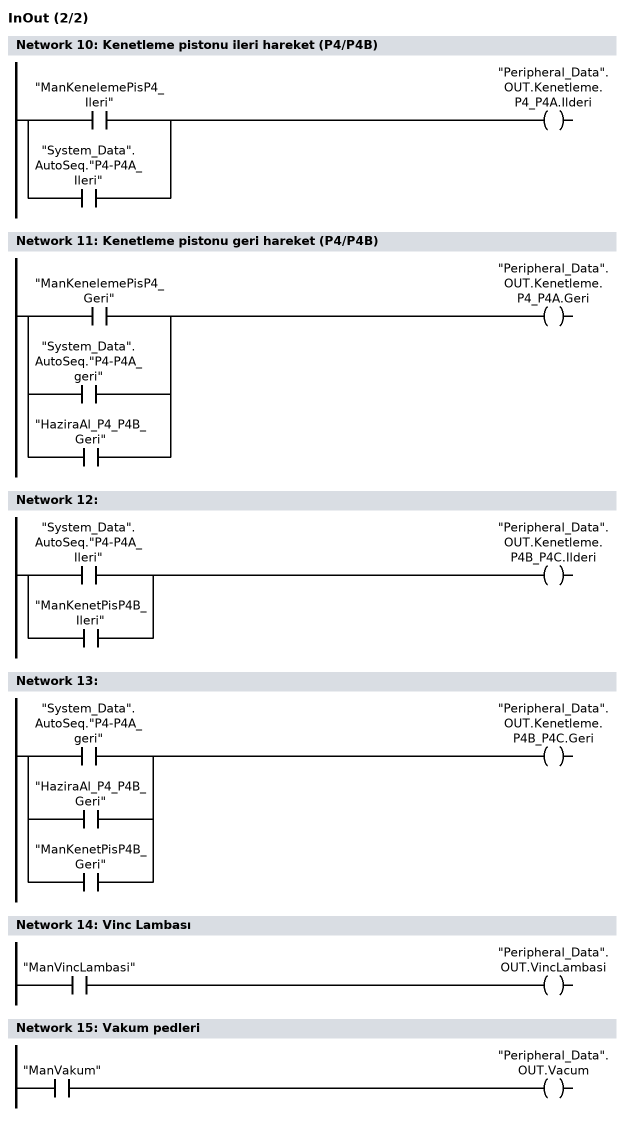
   RUNG wire#powerrail
      Contact( "ManKenelemePisP4_Ileri" )
      wire#w1
      Coil( "Peripheral_Data".OUT.Kenetleme.P4_P4A.Ilderi )
   END_RUNG
   RUNG wire#powerrail
      Contact( "System_Data".AutoSeq."P4-P4A_Ileri" )
   END_RUNG wire#w1
   // the same network as SCL:
   "Peripheral_Data".OUT.Kenetleme.P4_P4A.Ilderi := "ManKenelemePisP4_Ileri" OR "System_Data".AutoSeq."P4-P4A_Ileri";
END_REGION

REGION Network 11: Kenetleme pistonu geri hareket (P4/P4B)
   RUNG wire#powerrail
      Contact( "ManKenelemePisP4_Geri" )
      wire#w1
      Coil( "Peripheral_Data".OUT.Kenetleme.P4_P4A.Geri )
   END_RUNG
   RUNG wire#powerrail
      Contact( "System_Data".AutoSeq."P4-P4A_geri" )
   END_RUNG wire#w1
   RUNG wire#powerrail
      Contact( "HaziraAl_P4_P4B_Geri" )
   END_RUNG wire#w1
   // the same network as SCL:
   "Peripheral_Data".OUT.Kenetleme.P4_P4A.Geri := "ManKenelemePisP4_Geri" OR "System_Data".AutoSeq."P4-P4A_geri" OR "HaziraAl_P4_P4B_Geri";
END_REGION

REGION Network 12
   RUNG wire#powerrail
      Contact( "System_Data".AutoSeq."P4-P4A_Ileri" )
      wire#w1
      Coil( "Peripheral_Data".OUT.Kenetleme.P4B_P4C.Ilderi )
   END_RUNG
   RUNG wire#powerrail
      Contact( "ManKenetPisP4B_Ileri" )
   END_RUNG wire#w1
   // the same network as SCL:
   "Peripheral_Data".OUT.Kenetleme.P4B_P4C.Ilderi := "System_Data".AutoSeq."P4-P4A_Ileri" OR "ManKenetPisP4B_Ileri";
END_REGION

REGION Network 13
   RUNG wire#powerrail
      Contact( "System_Data".AutoSeq."P4-P4A_geri" )
      wire#w1
      Coil( "Peripheral_Data".OUT.Kenetleme.P4B_P4C.Geri )
   END_RUNG
   RUNG wire#powerrail
      Contact( "HaziraAl_P4_P4B_Geri" )
   END_RUNG wire#w1
   RUNG wire#powerrail
      Contact( "ManKenetPisP4B_Geri" )
   END_RUNG wire#w1
   // the same network as SCL:
   "Peripheral_Data".OUT.Kenetleme.P4B_P4C.Geri := "System_Data".AutoSeq."P4-P4A_geri" OR "HaziraAl_P4_P4B_Geri" OR "ManKenetPisP4B_Geri";
END_REGION

REGION Network 14: Vinc Lambası
   RUNG wire#powerrail
      Contact( "ManVincLambasi" )
      Coil( "Peripheral_Data".OUT.VincLambasi )
   END_RUNG
   // the same network as SCL:
   "Peripheral_Data".OUT.VincLambasi := "ManVincLambasi";
END_REGION

REGION Network 15: Vakum pedleri
   RUNG wire#powerrail
      Contact( "ManVakum" )
      Coil( "Peripheral_Data".OUT.Vacum )
   END_RUNG
   // the same network as SCL:
   "Peripheral_Data".OUT.Vacum := "ManVakum";
END_REGION
END_FUNCTION_BLOCK

FUNCTION "Peripheral" : Void   // FC2, SCL
{ S7_Optimized_Access := 'TRUE' }
VERSION : 0.1
BEGIN

   (**************************
   ******** INPUT *************
   **************************)

   "Peripheral_Data".IN.Acil_Stop := "I0.0";
   "Peripheral_Data".IN.CiftEl.IN1 := "I0.1";

   "Peripheral_Data".IN.CiftEl.IN2 := "I3.6";
   "Peripheral_Data".IN.CiftEl.IN3 := "I3.7";
   "Peripheral_Data".IN.VakumJen := "I0.2" OR "I0.3";

   "Peripheral_Data".IN.EnAyar.P1.Ileride := "I0.4";
   "Peripheral_Data".IN.EnAyar.P1.Geride := "I0.5";
   "Peripheral_Data".IN.EnAyar.P1A.Ileride := "I0.6";
   "Peripheral_Data".IN.EnAyar.P1A.Geride := "I0.7";

   "Peripheral_Data".IN.EnAyar.P2.Ileride := "I1.0";
   "Peripheral_Data".IN.EnAyar.P2.Geride := "I1.1";
   "Peripheral_Data".IN.EnAyar.P2A.Ileride := "I1.2";
   "Peripheral_Data".IN.EnAyar.P2A.Geride := "I1.3";

   "Peripheral_Data".IN.KademeAyar.P3.Ileride := "I1.4";
   "Peripheral_Data".IN.KademeAyar.P3.Geride := "I1.5";

   "Peripheral_Data".IN.Kenetleme.P4.Ilderide := "I2.0";
   "Peripheral_Data".IN.Kenetleme.P4.Geride := "I2.1";
   "Peripheral_Data".IN.Kenetleme.P4B.Ilderide := "I2.2";
   "Peripheral_Data".IN.Kenetleme.P4B.Geride := "I2.3";

   "Peripheral_Data".IN.VincUstuLamba := "I2.4";
   "Peripheral_Data".IN.ServoHomeSen := "I2.5";

   // "Peripheral_Data".IN.KademeAyar.P3A.Ileride := "I2.0";
   // "Peripheral_Data".IN.KademeAyar.P3A.Geride := "I2.1";

   // "Peripheral_Data".IN.Kenetleme.P4.Ilderide := "I2.2";
   // "Peripheral_Data".IN.Kenetleme.P4.Geride := "I2.3";
   // "Peripheral_Data".IN.Kenetleme.P4A.Ilderide := "I2.4";
   // "Peripheral_Data".IN.Kenetleme.P4A.Geride := "I2.5";

   // "Peripheral_Data".IN.Kenetleme.P4B.Ilderide := "I2.6";
   // "Peripheral_Data".IN.Kenetleme.P4B.Geride := "I2.7";
   // "Peripheral_Data".IN.Kenetleme.P4C.Ilderide := "I3.0";
   // "Peripheral_Data".IN.Kenetleme.P4C.Geride := "I3.1";

   // "Peripheral_Data".IN.VincUstuLamba := "I3.2";

   (**************************
   ******** OUTPUT ***********
   **************************)
   "Q0.0" := "Peripheral_Data".OUT.LAMBA.Kirmizi;
   "Q0.1" := "Peripheral_Data".OUT.LAMBA.Sari;
   "Q0.2" := "Peripheral_Data".OUT.LAMBA.Yesil;

   "Q0.3" := "Peripheral_Data".OUT.Vacum;
   "Q0.4" := "Peripheral_Data".OUT.VincLambasi;
   "Q0.5" := "Peripheral_Data".OUT.LAMBA.Buzzer;


   //*****************************************//
   //************* FESTO PROFINET ************//
   "Q4.0" := "Peripheral_Data".OUT.Kenetleme.P4B_P4C.Geri;
   "Q4.1" := "Peripheral_Data".OUT.Kenetleme.P4B_P4C.Ilderi;
   "Q4.2" := "Peripheral_Data".OUT.Kenetleme.P4_P4A.Geri;
   "Q4.3" := "Peripheral_Data".OUT.Kenetleme.P4_P4A.Ilderi;
   "Q4.4" := "Peripheral_Data".OUT.EnAyar.P1.Geri;
   "Q4.5" := "Peripheral_Data".OUT.EnAyar.P1.Ileri;
   "Q4.6" := "Peripheral_Data".OUT.EnAyar.P2.Geri;
   "Q4.7" := "Peripheral_Data".OUT.EnAyar.P2.Ileri;

   "Q5.0" := "Peripheral_Data".OUT.KademeAyar.P3.Geri;
   "Q5.1" := "Peripheral_Data".OUT.KademeAyar.P3.Ileri;
END_FUNCTION

FUNCTION "Station" : Void   // FC3, LAD
{ S7_Optimized_Access := 'TRUE' }
VERSION : 0.1
BEGIN

REGION Network 1: otomatik moda gecis
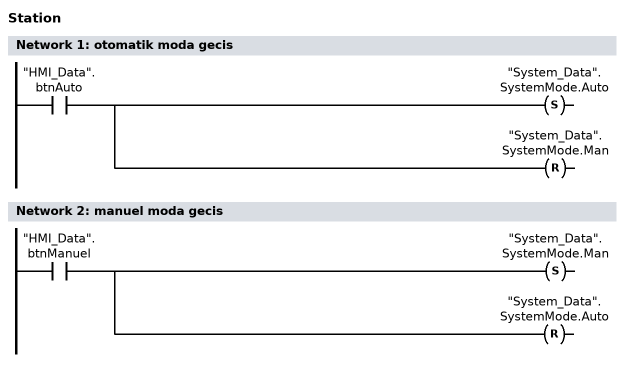
   RUNG wire#powerrail
      Contact( "HMI_Data".btnAuto )
      wire#w1
      S_Coil( "System_Data".SystemMode.Auto )
   END_RUNG
   RUNG wire#w1
      R_Coil( "System_Data".SystemMode.Man )
   END_RUNG
   // the same network as SCL:
   IF "HMI_Data".btnAuto THEN
       "System_Data".SystemMode.Auto := TRUE;
       "System_Data".SystemMode.Man := FALSE;
   END_IF;
END_REGION

REGION Network 2: manuel moda gecis
   RUNG wire#powerrail
      Contact( "HMI_Data".btnManuel )
      wire#w1
      S_Coil( "System_Data".SystemMode.Man )
   END_RUNG
   RUNG wire#w1
      R_Coil( "System_Data".SystemMode.Auto )
   END_RUNG
   // the same network as SCL:
   IF "HMI_Data".btnManuel THEN
       "System_Data".SystemMode.Man := TRUE;
       "System_Data".SystemMode.Auto := FALSE;
   END_IF;
END_REGION
END_FUNCTION

FUNCTION "HMI" : Void   // FC5, LAD
{ S7_Optimized_Access := 'TRUE' }
VERSION : 0.1
BEGIN

REGION Network 2 (SCL)
   // en ayar psitonu izleme 
   "HMI_Data".Status.EnAyarPis.P1.Ileride := "Peripheral_Data".IN.EnAyar.P1.Ileride
   AND "Peripheral_Data".IN.EnAyar.P1A.Ileride;
   "HMI_Data".Status.EnAyarPis.P2.Ileride := "Peripheral_Data".IN.EnAyar.P2.Ileride
   AND "Peripheral_Data".IN.EnAyar.P2A.Ileride;

   "HMI_Data".Status.EnAyarPis.P1.Geride := "Peripheral_Data".IN.EnAyar.P1.Geride
   AND "Peripheral_Data".IN.EnAyar.P1A.Geride;
   "HMI_Data".Status.EnAyarPis.P2.Geride := "Peripheral_Data".IN.EnAyar.P2.Geride
   AND "Peripheral_Data".IN.EnAyar.P2A.Geride;

   // kademe psitonu izleme 
   "HMI_Data".Status.KademePis_P3.Ileride := "Peripheral_Data".IN.KademeAyar.P3.Ileride;

   "HMI_Data".Status.KademePis_P3.Geride := "Peripheral_Data".IN.KademeAyar.P3.Geride;

   // kenetleme psitonu izleme
   "HMI_Data".Status.KenetlemePis_P4.Ileride := "Peripheral_Data".IN.Kenetleme.P4.Ilderide
   AND "Peripheral_Data".IN.Kenetleme.P4B.Ilderide;

   "HMI_Data".Status.KenetlemePis_P4.Geride := "Peripheral_Data".IN.Kenetleme.P4.Geride
   AND "Peripheral_Data".IN.Kenetleme.P4B.Geride;

   //Sistem secilen modele gore konumu hazir ise hazira al butonu yeşil olsun
   IF "Receipt".CurrentModel.Class = 0 THEN
       "System_Data".Ready := "ClassA_Hazir";
   ELSIF "Receipt".CurrentModel.Class = 1 THEN
       "System_Data".Ready := "ClassE_Hazir";
   ELSIF "Receipt".CurrentModel.Class = 2 THEN
       "System_Data".Ready := "ClassF_Hazir";
   ELSE
       "System_Data".Ready := false;
   END_IF;
END_REGION
END_FUNCTION

FUNCTION "UyariLambasi" : Void   // FC6, LAD
{ S7_Optimized_Access := 'TRUE' }
VERSION : 0.1
   VAR_TEMP
      wCheckAlarmWord : Word;   // "03FF" - piston timeout ve servo arıza bilgileri
      bCheckAlarmWord : Bool;
   END_VAR
BEGIN

REGION Network 1: Yesil lamba
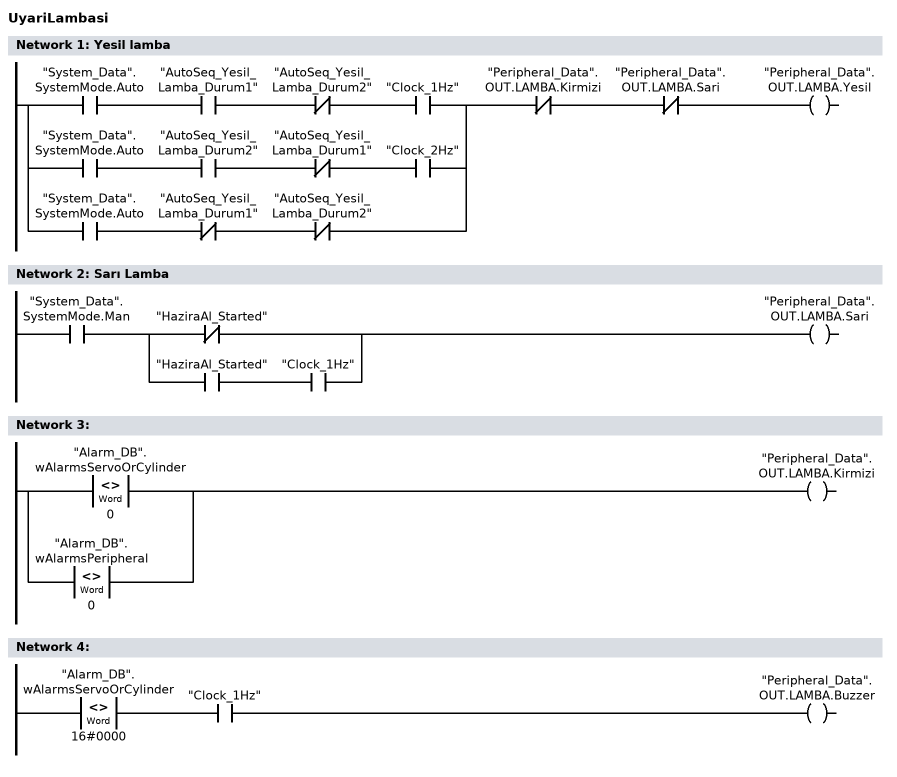
   RUNG wire#powerrail
      Contact( "System_Data".SystemMode.Auto )
      Contact( "AutoSeq_Yesil_Lamba_Durum1" )
      I_Contact( "AutoSeq_Yesil_Lamba_Durum2" )
      Contact( "Clock_1Hz" )
      wire#w1
      I_Contact( "Peripheral_Data".OUT.LAMBA.Kirmizi )
      I_Contact( "Peripheral_Data".OUT.LAMBA.Sari )
      Coil( "Peripheral_Data".OUT.LAMBA.Yesil )
   END_RUNG
   RUNG wire#powerrail
      Contact( "System_Data".SystemMode.Auto )
      Contact( "AutoSeq_Yesil_Lamba_Durum2" )
      I_Contact( "AutoSeq_Yesil_Lamba_Durum1" )
      Contact( "Clock_2Hz" )
   END_RUNG wire#w1
   RUNG wire#powerrail
      Contact( "System_Data".SystemMode.Auto )
      I_Contact( "AutoSeq_Yesil_Lamba_Durum1" )
      I_Contact( "AutoSeq_Yesil_Lamba_Durum2" )
   END_RUNG wire#w1
   // the same network as SCL:
   "Peripheral_Data".OUT.LAMBA.Yesil := (("System_Data".SystemMode.Auto AND "AutoSeq_Yesil_Lamba_Durum1" AND NOT "AutoSeq_Yesil_Lamba_Durum2" AND "Clock_1Hz") OR ("System_Data".SystemMode.Auto AND "AutoSeq_Yesil_Lamba_Durum2" AND NOT "AutoSeq_Yesil_Lamba_Durum1" AND "Clock_2Hz") OR ("System_Data".SystemMode.Auto AND NOT "AutoSeq_Yesil_Lamba_Durum1" AND NOT "AutoSeq_Yesil_Lamba_Durum2")) AND NOT "Peripheral_Data".OUT.LAMBA.Kirmizi AND NOT "Peripheral_Data".OUT.LAMBA.Sari;
END_REGION

REGION Network 2: Sarı Lamba
   RUNG wire#powerrail
      Contact( "System_Data".SystemMode.Man )
      wire#w1
      I_Contact( "HaziraAl_Started" )
      wire#w2
      Coil( "Peripheral_Data".OUT.LAMBA.Sari )
   END_RUNG
   RUNG wire#w1
      Contact( "HaziraAl_Started" )
      Contact( "Clock_1Hz" )
   END_RUNG wire#w2
   // the same network as SCL:
   "Peripheral_Data".OUT.LAMBA.Sari := "System_Data".SystemMode.Man AND (NOT "HaziraAl_Started" OR ("HaziraAl_Started" AND "Clock_1Hz"));
END_REGION

REGION Network 3
   RUNG wire#powerrail
      { S7_Templates := "SrcType := Word" } NE_Contact(in1 := "Alarm_DB".wAlarmsServoOrCylinder, in2 := 0)
      wire#w1
      Coil( "Peripheral_Data".OUT.LAMBA.Kirmizi )
   END_RUNG
   RUNG wire#powerrail
      { S7_Templates := "SrcType := Word" } NE_Contact(in1 := "Alarm_DB".wAlarmsPeripheral, in2 := 0)
   END_RUNG wire#w1
   // the same network as SCL:
   "Peripheral_Data".OUT.LAMBA.Kirmizi := ("Alarm_DB".wAlarmsServoOrCylinder <> 0) OR ("Alarm_DB".wAlarmsPeripheral <> 0);
END_REGION

REGION Network 4
   RUNG wire#powerrail
      { S7_Templates := "SrcType := Word" } NE_Contact(in1 := "Alarm_DB".wAlarmsServoOrCylinder, in2 := 16#0000)
      Contact( "Clock_1Hz" )
      Coil( "Peripheral_Data".OUT.LAMBA.Buzzer )
   END_RUNG
   // the same network as SCL:
   "Peripheral_Data".OUT.LAMBA.Buzzer := ("Alarm_DB".wAlarmsServoOrCylinder <> 16#0000) AND "Clock_1Hz";
END_REGION
END_FUNCTION

// folder: Manuel

FUNCTION_BLOCK "Manuel"   // FB3, LAD
{ S7_Optimized_Access := 'TRUE' }
VERSION : 0.1
   VAR_TEMP   // added for the SCL form of the ladder/FBD networks
      _w1 : Bool;
   END_VAR
BEGIN

REGION Network 1: Servo Manuel Jog 1
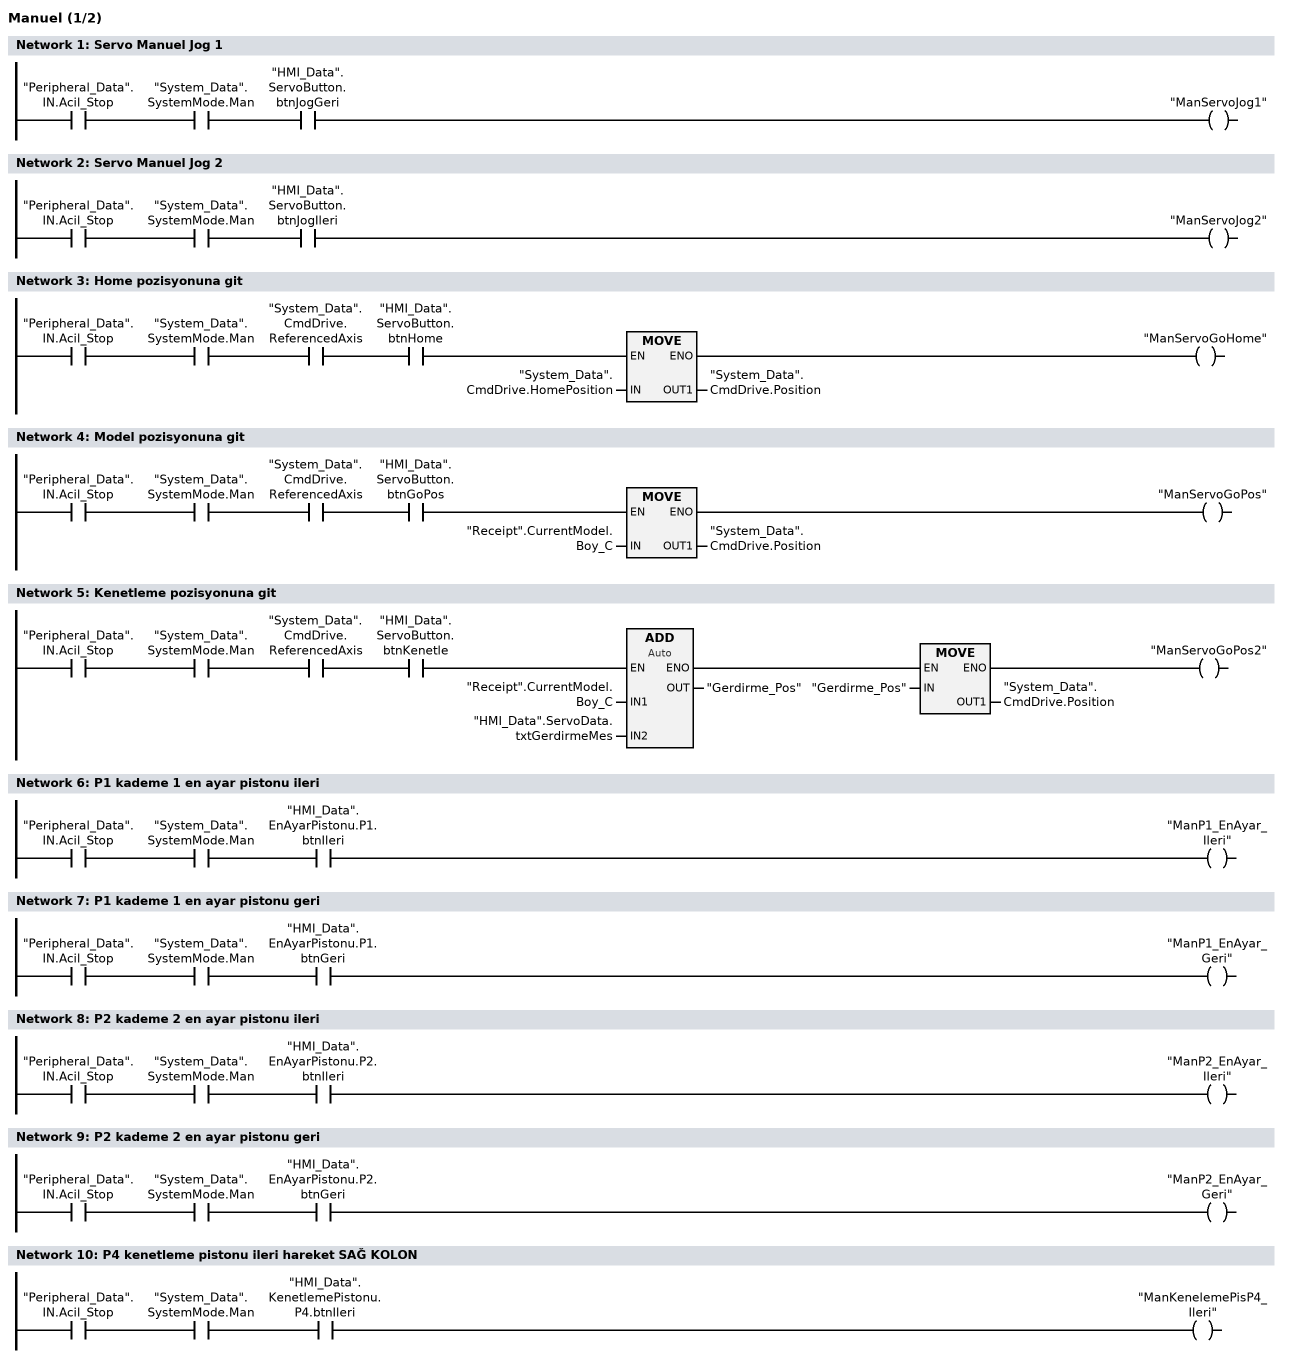
   RUNG wire#powerrail
      Contact( "Peripheral_Data".IN.Acil_Stop )
      Contact( "System_Data".SystemMode.Man )
      Contact( "HMI_Data".ServoButton.btnJogGeri )
      Coil( "ManServoJog1" )
   END_RUNG
   // the same network as SCL:
   "ManServoJog1" := "Peripheral_Data".IN.Acil_Stop AND "System_Data".SystemMode.Man AND "HMI_Data".ServoButton.btnJogGeri;
END_REGION

REGION Network 2: Servo Manuel Jog 2
   RUNG wire#powerrail
      Contact( "Peripheral_Data".IN.Acil_Stop )
      Contact( "System_Data".SystemMode.Man )
      Contact( "HMI_Data".ServoButton.btnJogIleri )
      Coil( "ManServoJog2" )
   END_RUNG
   // the same network as SCL:
   "ManServoJog2" := "Peripheral_Data".IN.Acil_Stop AND "System_Data".SystemMode.Man AND "HMI_Data".ServoButton.btnJogIleri;
END_REGION

REGION Network 3: Home pozisyonuna git
   RUNG wire#powerrail
      Contact( "Peripheral_Data".IN.Acil_Stop )
      Contact( "System_Data".SystemMode.Man )
      Contact( "System_Data".CmdDrive.ReferencedAxis )
      Contact( "HMI_Data".ServoButton.btnHome )
      Move(in := "System_Data".CmdDrive.HomePosition, out1 => "System_Data".CmdDrive.Position)
      Coil( "ManServoGoHome" )
   END_RUNG
   // the same network as SCL:
   #_w1 := "Peripheral_Data".IN.Acil_Stop AND "System_Data".SystemMode.Man AND "System_Data".CmdDrive.ReferencedAxis AND "HMI_Data".ServoButton.btnHome;
   IF #_w1 THEN "System_Data".CmdDrive.Position := "System_Data".CmdDrive.HomePosition; END_IF;
   "ManServoGoHome" := #_w1;
END_REGION

REGION Network 4: Model pozisyonuna git
   RUNG wire#powerrail
      Contact( "Peripheral_Data".IN.Acil_Stop )
      Contact( "System_Data".SystemMode.Man )
      Contact( "System_Data".CmdDrive.ReferencedAxis )
      Contact( "HMI_Data".ServoButton.btnGoPos )
      Move(in := "Receipt".CurrentModel.Boy_C, out1 => "System_Data".CmdDrive.Position)
      Coil( "ManServoGoPos" )
   END_RUNG
   // the same network as SCL:
   #_w1 := "Peripheral_Data".IN.Acil_Stop AND "System_Data".SystemMode.Man AND "System_Data".CmdDrive.ReferencedAxis AND "HMI_Data".ServoButton.btnGoPos;
   IF #_w1 THEN "System_Data".CmdDrive.Position := "Receipt".CurrentModel.Boy_C; END_IF;
   "ManServoGoPos" := #_w1;
END_REGION

REGION Network 5: Kenetleme pozisyonuna git
   RUNG wire#powerrail
      Contact( "Peripheral_Data".IN.Acil_Stop )
      Contact( "System_Data".SystemMode.Man )
      Contact( "System_Data".CmdDrive.ReferencedAxis )
      Contact( "HMI_Data".ServoButton.btnKenetle )
      Add(in1 := "Receipt".CurrentModel.Boy_C, in2 := "HMI_Data".ServoData.txtGerdirmeMes, out => "Gerdirme_Pos")
      Move(in := "Gerdirme_Pos", out1 => "System_Data".CmdDrive.Position)
      Coil( "ManServoGoPos2" )
   END_RUNG
   // the same network as SCL:
   #_w1 := "Peripheral_Data".IN.Acil_Stop AND "System_Data".SystemMode.Man AND "System_Data".CmdDrive.ReferencedAxis AND "HMI_Data".ServoButton.btnKenetle;
   IF #_w1 THEN
       "Gerdirme_Pos" := "Receipt".CurrentModel.Boy_C + "HMI_Data".ServoData.txtGerdirmeMes;
       "System_Data".CmdDrive.Position := "Gerdirme_Pos";
   END_IF;
   "ManServoGoPos2" := #_w1;
END_REGION

REGION Network 6: P1 kademe 1 en ayar pistonu ileri
   RUNG wire#powerrail
      Contact( "Peripheral_Data".IN.Acil_Stop )
      Contact( "System_Data".SystemMode.Man )
      Contact( "HMI_Data".EnAyarPistonu.P1.btnIleri )
      Coil( "ManP1_EnAyar_Ileri" )
   END_RUNG
   // the same network as SCL:
   "ManP1_EnAyar_Ileri" := "Peripheral_Data".IN.Acil_Stop AND "System_Data".SystemMode.Man AND "HMI_Data".EnAyarPistonu.P1.btnIleri;
END_REGION

REGION Network 7: P1 kademe 1 en ayar pistonu geri
   RUNG wire#powerrail
      Contact( "Peripheral_Data".IN.Acil_Stop )
      Contact( "System_Data".SystemMode.Man )
      Contact( "HMI_Data".EnAyarPistonu.P1.btnGeri )
      Coil( "ManP1_EnAyar_Geri" )
   END_RUNG
   // the same network as SCL:
   "ManP1_EnAyar_Geri" := "Peripheral_Data".IN.Acil_Stop AND "System_Data".SystemMode.Man AND "HMI_Data".EnAyarPistonu.P1.btnGeri;
END_REGION

REGION Network 8: P2 kademe 2 en ayar pistonu ileri
   RUNG wire#powerrail
      Contact( "Peripheral_Data".IN.Acil_Stop )
      Contact( "System_Data".SystemMode.Man )
      Contact( "HMI_Data".EnAyarPistonu.P2.btnIleri )
      Coil( "ManP2_EnAyar_Ileri" )
   END_RUNG
   // the same network as SCL:
   "ManP2_EnAyar_Ileri" := "Peripheral_Data".IN.Acil_Stop AND "System_Data".SystemMode.Man AND "HMI_Data".EnAyarPistonu.P2.btnIleri;
END_REGION

REGION Network 9: P2 kademe 2 en ayar pistonu geri
   RUNG wire#powerrail
      Contact( "Peripheral_Data".IN.Acil_Stop )
      Contact( "System_Data".SystemMode.Man )
      Contact( "HMI_Data".EnAyarPistonu.P2.btnGeri )
      Coil( "ManP2_EnAyar_Geri" )
   END_RUNG
   // the same network as SCL:
   "ManP2_EnAyar_Geri" := "Peripheral_Data".IN.Acil_Stop AND "System_Data".SystemMode.Man AND "HMI_Data".EnAyarPistonu.P2.btnGeri;
END_REGION

REGION Network 10: P4 kenetleme pistonu ileri hareket SAĞ KOLON
   RUNG wire#powerrail
      Contact( "Peripheral_Data".IN.Acil_Stop )
      Contact( "System_Data".SystemMode.Man )
      Contact( "HMI_Data".KenetlemePistonu.P4.btnIleri )
      Coil( "ManKenelemePisP4_Ileri" )
   END_RUNG
   // the same network as SCL:
   "ManKenelemePisP4_Ileri" := "Peripheral_Data".IN.Acil_Stop AND "System_Data".SystemMode.Man AND "HMI_Data".KenetlemePistonu.P4.btnIleri;
END_REGION

REGION Network 11: P4 kenetleme pistonu geri hareket (SAĞ KOLON)
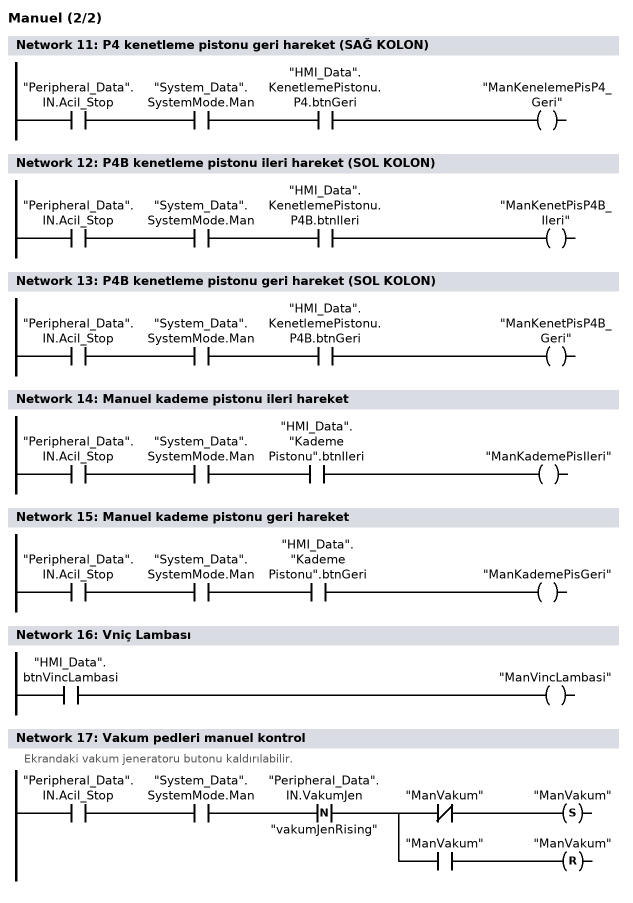
   RUNG wire#powerrail
      Contact( "Peripheral_Data".IN.Acil_Stop )
      Contact( "System_Data".SystemMode.Man )
      Contact( "HMI_Data".KenetlemePistonu.P4.btnGeri )
      Coil( "ManKenelemePisP4_Geri" )
   END_RUNG
   // the same network as SCL:
   "ManKenelemePisP4_Geri" := "Peripheral_Data".IN.Acil_Stop AND "System_Data".SystemMode.Man AND "HMI_Data".KenetlemePistonu.P4.btnGeri;
END_REGION

REGION Network 12: P4B kenetleme pistonu ileri hareket (SOL KOLON)
   RUNG wire#powerrail
      Contact( "Peripheral_Data".IN.Acil_Stop )
      Contact( "System_Data".SystemMode.Man )
      Contact( "HMI_Data".KenetlemePistonu.P4B.btnIleri )
      Coil( "ManKenetPisP4B_Ileri" )
   END_RUNG
   // the same network as SCL:
   "ManKenetPisP4B_Ileri" := "Peripheral_Data".IN.Acil_Stop AND "System_Data".SystemMode.Man AND "HMI_Data".KenetlemePistonu.P4B.btnIleri;
END_REGION

REGION Network 13: P4B kenetleme pistonu geri hareket (SOL KOLON)
   RUNG wire#powerrail
      Contact( "Peripheral_Data".IN.Acil_Stop )
      Contact( "System_Data".SystemMode.Man )
      Contact( "HMI_Data".KenetlemePistonu.P4B.btnGeri )
      Coil( "ManKenetPisP4B_Geri" )
   END_RUNG
   // the same network as SCL:
   "ManKenetPisP4B_Geri" := "Peripheral_Data".IN.Acil_Stop AND "System_Data".SystemMode.Man AND "HMI_Data".KenetlemePistonu.P4B.btnGeri;
END_REGION

REGION Network 14: Manuel kademe pistonu ileri hareket
   RUNG wire#powerrail
      Contact( "Peripheral_Data".IN.Acil_Stop )
      Contact( "System_Data".SystemMode.Man )
      Contact( "HMI_Data"."Kademe Pistonu".btnIleri )
      Coil( "ManKademePisIleri" )
   END_RUNG
   // the same network as SCL:
   "ManKademePisIleri" := "Peripheral_Data".IN.Acil_Stop AND "System_Data".SystemMode.Man AND "HMI_Data"."Kademe Pistonu".btnIleri;
END_REGION

REGION Network 15: Manuel kademe pistonu geri hareket
   RUNG wire#powerrail
      Contact( "Peripheral_Data".IN.Acil_Stop )
      Contact( "System_Data".SystemMode.Man )
      Contact( "HMI_Data"."Kademe Pistonu".btnGeri )
      Coil( "ManKademePisGeri" )
   END_RUNG
   // the same network as SCL:
   "ManKademePisGeri" := "Peripheral_Data".IN.Acil_Stop AND "System_Data".SystemMode.Man AND "HMI_Data"."Kademe Pistonu".btnGeri;
END_REGION

REGION Network 16: Vniç Lambası
   RUNG wire#powerrail
      Contact( "HMI_Data".btnVincLambasi )
      Coil( "ManVincLambasi" )
   END_RUNG
   // the same network as SCL:
   "ManVincLambasi" := "HMI_Data".btnVincLambasi;
END_REGION

REGION Network 17: Vakum pedleri manuel kontrol
   // Ekrandaki vakum jeneratoru butonu kaldırılabilir.
   RUNG wire#powerrail
      Contact( "Peripheral_Data".IN.Acil_Stop )
      Contact( "System_Data".SystemMode.Man )
      N_Contact(operand := "Peripheral_Data".IN.VakumJen, bit := "vakumJenRising")
      wire#w1
      I_Contact( "ManVakum" )
      S_Coil( "ManVakum" )
   END_RUNG
   RUNG wire#w1
      Contact( "ManVakum" )
      R_Coil( "ManVakum" )
   END_RUNG
   // the same network as SCL:
   #_w1 := "Peripheral_Data".IN.Acil_Stop AND "System_Data".SystemMode.Man AND NOT "Peripheral_Data".IN.VakumJen AND "vakumJenRising";   // falling edge of "Peripheral_Data".IN.VakumJen
   "vakumJenRising" := "Peripheral_Data".IN.VakumJen;
   IF #_w1 AND NOT "ManVakum" THEN "ManVakum" := TRUE; END_IF;
   IF #_w1 AND "ManVakum" THEN "ManVakum" := FALSE; END_IF;
END_REGION
END_FUNCTION_BLOCK

// folder: Otomatik

FUNCTION_BLOCK "Otomatik_Seq_LAD"   // FB5, LAD
{ S7_Optimized_Access := 'TRUE' }
VERSION : 0.1
   VAR_INPUT
      Start : Bool;
      Stop : Bool;
      EmergencyStop : Bool;
   END_VAR
   VAR_OUTPUT
      Busy : Bool;
      Done : Bool;
      Message : String[50];
   END_VAR
   VAR
      MessageDelay_Instance : TON_TIME;
      Adim2_Pos_Delay : TON_TIME;
      IEC_Timer_0_Instance : TON_TIME;
      IEC_Timer_0_Instance_1 : TON_TIME;
      IEC_Timer_0_Instance_2 : TON_TIME;
      KenetlemeTimer_Instance : TON_TIME;
   END_VAR
   VAR_TEMP
      bStart : Bool;
      bEmergencyStop : Bool;
      bStop : Bool;
      bHazir : Bool;
   END_VAR
   VAR CONSTANT
      eIDLE : Int;
      eCHECK_CLASS : Int := 1;
      eKENETLE : Int := 2;
      eKENETLE_2 : Int := 8;
      eCLASS_A_2 : Int := 9;
      eCLASS_E : Int := 3;
      eCLASS_F : Int := 4;
      eSUCCES : Int := 5;
      eERROR : Int := 6;
      eACILSTOP : Int := 7;
      ePAUSE : Int := 10;
      eFREE : Int := 11;
      eACIL : Int := 12;
      eCHECK_P3 : Int := 13;
      eP4_Kenetle : Int := 14;
   END_VAR
   VAR_TEMP   // added for the SCL form of the ladder/FBD networks
      _w1 : Bool;
   END_VAR
BEGIN

REGION Network 2
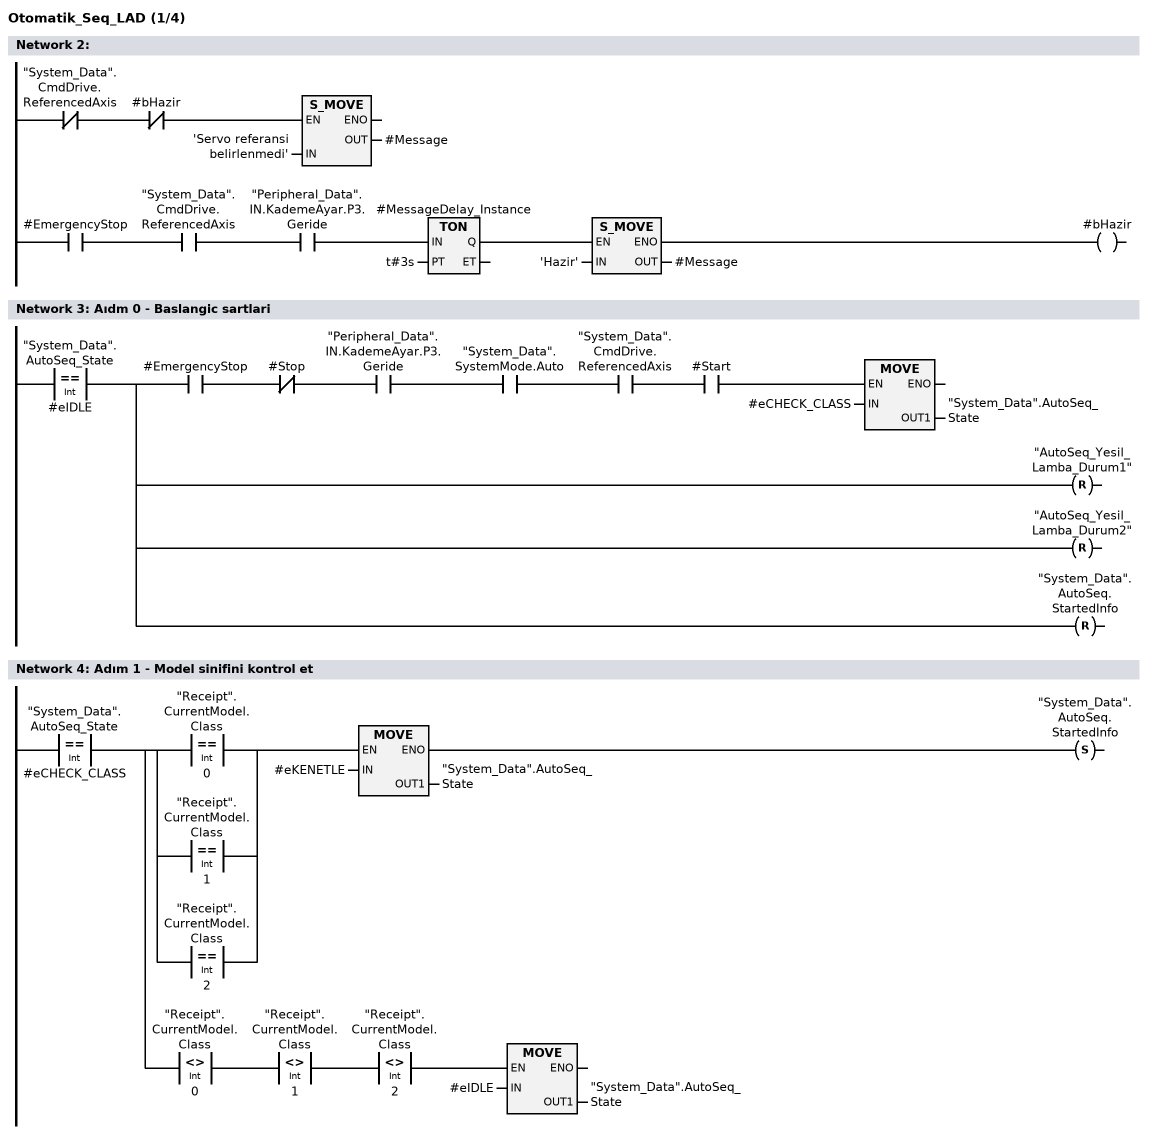
   IF NOT "System_Data".CmdDrive.ReferencedAxis AND NOT #bHazir THEN
       #Message := 'Servo referansi belirlenmedi';
   END_IF;
   #MessageDelay_Instance(IN := #EmergencyStop AND "System_Data".CmdDrive.ReferencedAxis AND "Peripheral_Data".IN.KademeAyar.P3.Geride,   // TON
                          PT := t#3s);
   IF #MessageDelay_Instance.Q THEN #Message := 'Hazir'; END_IF;
   #bHazir := #MessageDelay_Instance.Q;
END_REGION

REGION Network 3: Aıdm 0 - Baslangic sartlari
   RUNG wire#powerrail
      { S7_Templates := "SrcType := Int" } EQ_Contact(in1 := "System_Data".AutoSeq_State, in2 := #eIDLE)
      wire#w1
      Contact( #EmergencyStop )
      I_Contact( #Stop )
      Contact( "Peripheral_Data".IN.KademeAyar.P3.Geride )
      Contact( "System_Data".SystemMode.Auto )
      Contact( "System_Data".CmdDrive.ReferencedAxis )
      Contact( #Start )
      Move(in := #eCHECK_CLASS, out1 => "System_Data".AutoSeq_State)
   END_RUNG
   RUNG wire#w1
      R_Coil( "AutoSeq_Yesil_Lamba_Durum1" )
   END_RUNG
   RUNG wire#w1
      R_Coil( "AutoSeq_Yesil_Lamba_Durum2" )
   END_RUNG
   RUNG wire#w1
      R_Coil( "System_Data".AutoSeq.StartedInfo )
   END_RUNG
   // the same network as SCL:
   #_w1 := "System_Data".AutoSeq_State = #eIDLE;
   IF #_w1 AND #EmergencyStop AND NOT #Stop AND "Peripheral_Data".IN.KademeAyar.P3.Geride AND "System_Data".SystemMode.Auto AND "System_Data".CmdDrive.ReferencedAxis AND #Start THEN
       "System_Data".AutoSeq_State := #eCHECK_CLASS;
   END_IF;
   IF #_w1 THEN
       "AutoSeq_Yesil_Lamba_Durum1" := FALSE;
       "AutoSeq_Yesil_Lamba_Durum2" := FALSE;
       "System_Data".AutoSeq.StartedInfo := FALSE;
   END_IF;
END_REGION

REGION Network 4: Adım 1 - Model sinifini kontrol et
   RUNG wire#powerrail
      { S7_Templates := "SrcType := Int" } EQ_Contact(in1 := "System_Data".AutoSeq_State, in2 := #eCHECK_CLASS)
      wire#w1
      { S7_Templates := "SrcType := Int" } EQ_Contact(in1 := "Receipt".CurrentModel.Class, in2 := 0)
      wire#w2
      Move(in := #eKENETLE, out1 => "System_Data".AutoSeq_State)
      S_Coil( "System_Data".AutoSeq.StartedInfo )
   END_RUNG
   RUNG wire#w1
      { S7_Templates := "SrcType := Int" } EQ_Contact(in1 := "Receipt".CurrentModel.Class, in2 := 1)
   END_RUNG wire#w2
   RUNG wire#w1
      { S7_Templates := "SrcType := Int" } EQ_Contact(in1 := "Receipt".CurrentModel.Class, in2 := 2)
   END_RUNG wire#w2
   RUNG wire#w1
      { S7_Templates := "SrcType := Int" } NE_Contact(in1 := "Receipt".CurrentModel.Class, in2 := 0)
      { S7_Templates := "SrcType := Int" } NE_Contact(in1 := "Receipt".CurrentModel.Class, in2 := 1)
      { S7_Templates := "SrcType := Int" } NE_Contact(in1 := "Receipt".CurrentModel.Class, in2 := 2)
      Move(in := #eIDLE, out1 => "System_Data".AutoSeq_State)
   END_RUNG
   // the same network as SCL:
   #_w1 := "System_Data".AutoSeq_State = #eCHECK_CLASS;
   IF #_w1 AND (("Receipt".CurrentModel.Class = 0) OR ("Receipt".CurrentModel.Class = 1) OR ("Receipt".CurrentModel.Class = 2)) THEN
       "System_Data".AutoSeq_State := #eKENETLE;
       "System_Data".AutoSeq.StartedInfo := TRUE;
   END_IF;
   IF #_w1 AND ("Receipt".CurrentModel.Class <> 0) AND ("Receipt".CurrentModel.Class <> 1) AND ("Receipt".CurrentModel.Class <> 2) THEN
       "System_Data".AutoSeq_State := #eIDLE;
   END_IF;
END_REGION

REGION Network 5: Adım 2 - servo gerdirme konumuna ilerle
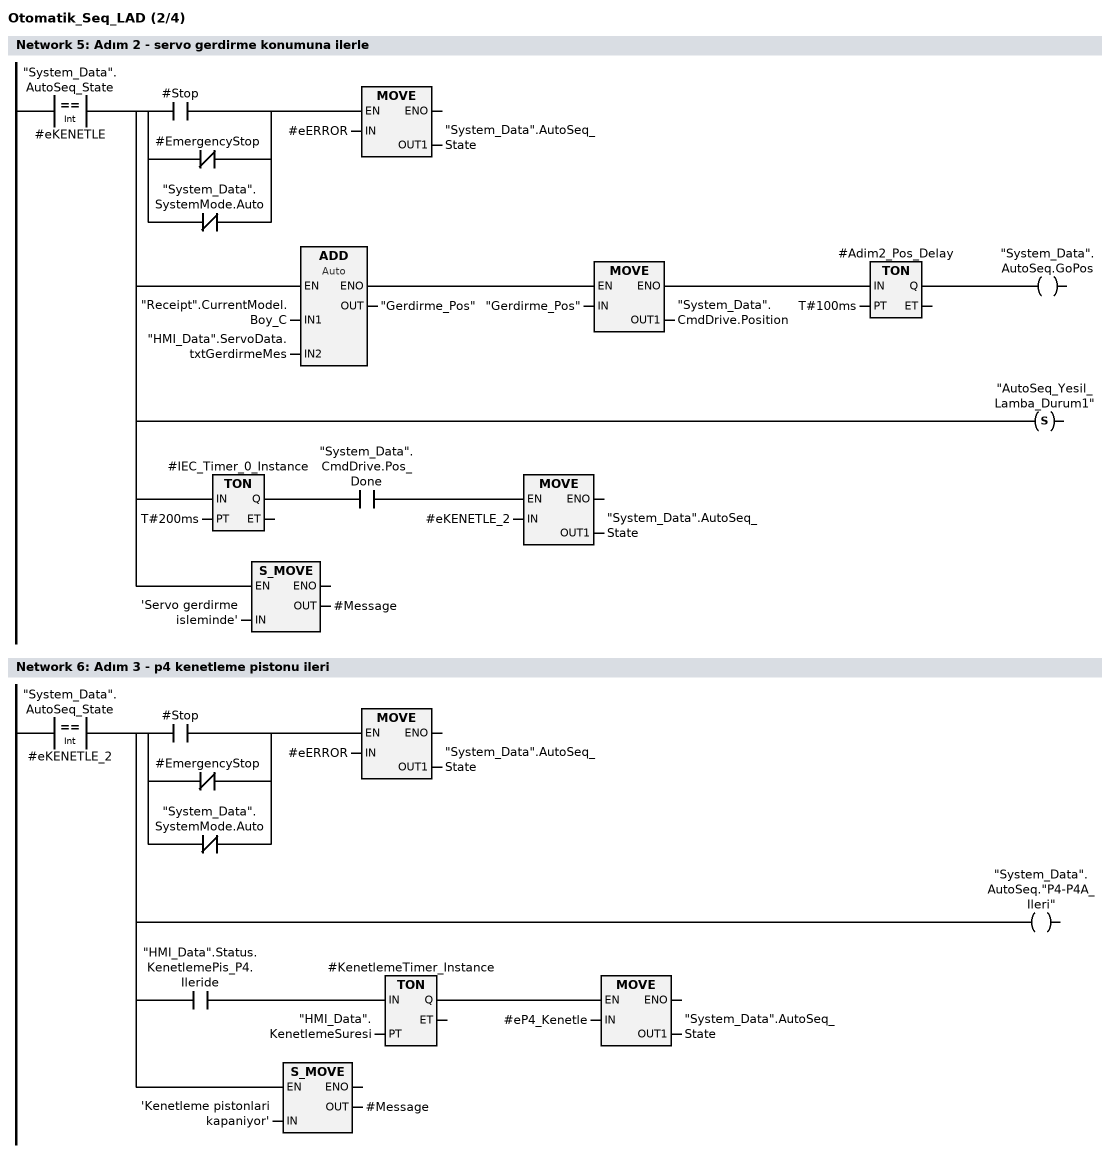
   #_w1 := "System_Data".AutoSeq_State = #eKENETLE;
   IF #_w1 AND (#Stop OR NOT #EmergencyStop OR NOT "System_Data".SystemMode.Auto) THEN
       "System_Data".AutoSeq_State := #eERROR;
   END_IF;
   IF #_w1 THEN
       "Gerdirme_Pos" := "Receipt".CurrentModel.Boy_C + "HMI_Data".ServoData.txtGerdirmeMes;
       "System_Data".CmdDrive.Position := "Gerdirme_Pos";
   END_IF;
   #Adim2_Pos_Delay(IN := #_w1, PT := T#100ms);   // TON
   "System_Data".AutoSeq.GoPos := #Adim2_Pos_Delay.Q;
   IF #_w1 THEN "AutoSeq_Yesil_Lamba_Durum1" := TRUE; END_IF;
   #IEC_Timer_0_Instance(IN := #_w1, PT := T#200ms);   // TON
   IF #IEC_Timer_0_Instance.Q AND "System_Data".CmdDrive.Pos_Done THEN
       "System_Data".AutoSeq_State := #eKENETLE_2;
   END_IF;
   IF #_w1 THEN #Message := 'Servo gerdirme isleminde'; END_IF;
END_REGION

REGION Network 6: Adım 3 - p4 kenetleme pistonu ileri
   #_w1 := "System_Data".AutoSeq_State = #eKENETLE_2;
   IF #_w1 AND (#Stop OR NOT #EmergencyStop OR NOT "System_Data".SystemMode.Auto) THEN
       "System_Data".AutoSeq_State := #eERROR;
   END_IF;
   "System_Data".AutoSeq."P4-P4A_Ileri" := #_w1;
   #KenetlemeTimer_Instance(IN := #_w1 AND "HMI_Data".Status.KenetlemePis_P4.Ileride,   // TON
                           PT := "HMI_Data".KenetlemeSuresi);
   IF #KenetlemeTimer_Instance.Q THEN "System_Data".AutoSeq_State := #eP4_Kenetle; END_IF;
   IF #_w1 THEN #Message := 'Kenetleme pistonlari kapaniyor'; END_IF;
END_REGION

REGION Network 7: p4 kenetleme pistonu geri ve p3 pistonu ileri
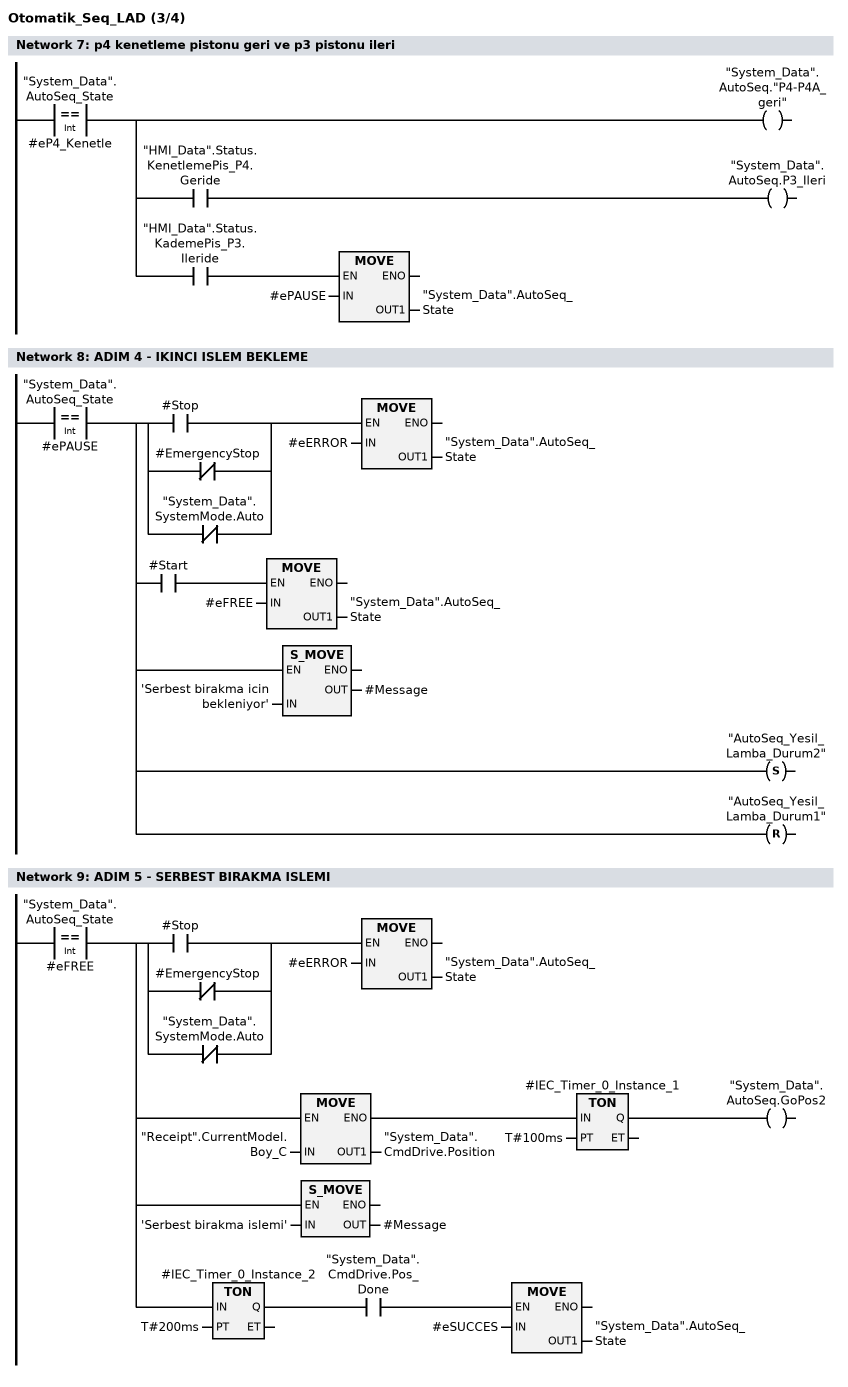
   RUNG wire#powerrail
      { S7_Templates := "SrcType := Int" } EQ_Contact(in1 := "System_Data".AutoSeq_State, in2 := #eP4_Kenetle)
      wire#w1
      Coil( "System_Data".AutoSeq."P4-P4A_geri" )
   END_RUNG
   RUNG wire#w1
      Contact( "HMI_Data".Status.KenetlemePis_P4.Geride )
      Coil( "System_Data".AutoSeq.P3_Ileri )
   END_RUNG
   RUNG wire#w1
      Contact( "HMI_Data".Status.KademePis_P3.Ileride )
      Move(in := #ePAUSE, out1 => "System_Data".AutoSeq_State)
   END_RUNG
   // the same network as SCL:
   "System_Data".AutoSeq."P4-P4A_geri" := "System_Data".AutoSeq_State = #eP4_Kenetle;
   "System_Data".AutoSeq.P3_Ileri := "System_Data".AutoSeq."P4-P4A_geri" AND "HMI_Data".Status.KenetlemePis_P4.Geride;
   IF "System_Data".AutoSeq."P4-P4A_geri" AND "HMI_Data".Status.KademePis_P3.Ileride THEN
       "System_Data".AutoSeq_State := #ePAUSE;
   END_IF;
END_REGION

REGION Network 8: ADIM 4 - IKINCI ISLEM BEKLEME
   RUNG wire#powerrail
      { S7_Templates := "SrcType := Int" } EQ_Contact(in1 := "System_Data".AutoSeq_State, in2 := #ePAUSE)
      wire#w1
      Contact( #Stop )
      wire#w2
      Move(in := #eERROR, out1 => "System_Data".AutoSeq_State)
   END_RUNG
   RUNG wire#w1
      I_Contact( #EmergencyStop )
   END_RUNG wire#w2
   RUNG wire#w1
      I_Contact( "System_Data".SystemMode.Auto )
   END_RUNG wire#w2
   RUNG wire#w1
      Contact( #Start )
      Move(in := #eFREE, out1 => "System_Data".AutoSeq_State)
   END_RUNG
   RUNG wire#w1
      S_Move(in := 'Serbest birakma icin bekleniyor', out => #Message)
   END_RUNG
   RUNG wire#w1
      S_Coil( "AutoSeq_Yesil_Lamba_Durum2" )
   END_RUNG
   RUNG wire#w1
      R_Coil( "AutoSeq_Yesil_Lamba_Durum1" )
   END_RUNG
   // the same network as SCL:
   #_w1 := "System_Data".AutoSeq_State = #ePAUSE;
   IF #_w1 AND (#Stop OR NOT #EmergencyStop OR NOT "System_Data".SystemMode.Auto) THEN
       "System_Data".AutoSeq_State := #eERROR;
   END_IF;
   IF #_w1 AND #Start THEN "System_Data".AutoSeq_State := #eFREE; END_IF;
   IF #_w1 THEN
       #Message := 'Serbest birakma icin bekleniyor';
       "AutoSeq_Yesil_Lamba_Durum2" := TRUE;
       "AutoSeq_Yesil_Lamba_Durum1" := FALSE;
   END_IF;
END_REGION

REGION Network 9: ADIM 5 - SERBEST BIRAKMA ISLEMI
   #_w1 := "System_Data".AutoSeq_State = #eFREE;
   IF #_w1 AND (#Stop OR NOT #EmergencyStop OR NOT "System_Data".SystemMode.Auto) THEN
       "System_Data".AutoSeq_State := #eERROR;
   END_IF;
   IF #_w1 THEN "System_Data".CmdDrive.Position := "Receipt".CurrentModel.Boy_C; END_IF;
   #IEC_Timer_0_Instance_1(IN := #_w1, PT := T#100ms);   // TON
   "System_Data".AutoSeq.GoPos2 := #IEC_Timer_0_Instance_1.Q;
   IF #_w1 THEN #Message := 'Serbest birakma islemi'; END_IF;
   #IEC_Timer_0_Instance_2(IN := #_w1, PT := T#200ms);   // TON
   IF #IEC_Timer_0_Instance_2.Q AND "System_Data".CmdDrive.Pos_Done THEN
       "System_Data".AutoSeq_State := #eSUCCES;
   END_IF;
END_REGION

REGION Network 10: ADIMLAR BASARILI ISE
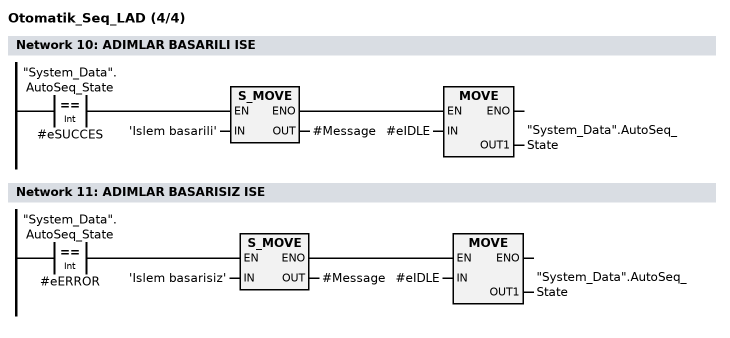
   RUNG wire#powerrail
      { S7_Templates := "SrcType := Int" } EQ_Contact(in1 := "System_Data".AutoSeq_State, in2 := #eSUCCES)
      S_Move(in := 'Islem basarili', out => #Message)
      Move(in := #eIDLE, out1 => "System_Data".AutoSeq_State)
   END_RUNG
   // the same network as SCL:
   IF "System_Data".AutoSeq_State = #eSUCCES THEN
       #Message := 'Islem basarili';
       "System_Data".AutoSeq_State := #eIDLE;
   END_IF;
END_REGION

REGION Network 11: ADIMLAR BASARISIZ ISE
   RUNG wire#powerrail
      { S7_Templates := "SrcType := Int" } EQ_Contact(in1 := "System_Data".AutoSeq_State, in2 := #eERROR)
      S_Move(in := 'Islem basarisiz', out => #Message)
      Move(in := #eIDLE, out1 => "System_Data".AutoSeq_State)
   END_RUNG
   // the same network as SCL:
   IF "System_Data".AutoSeq_State = #eERROR THEN
       #Message := 'Islem basarisiz';
       "System_Data".AutoSeq_State := #eIDLE;
   END_IF;
END_REGION
END_FUNCTION_BLOCK

FUNCTION "HaziraAl" : Void   // FC4, LAD
{ S7_Optimized_Access := 'TRUE' }
VERSION : 0.1
   VAR_INPUT
      Execute : Bool;   // Islemi yurut
      EmergencyStop : Bool;   // Acil stop
      IsServoPosDone : Bool;   // Servo konumu tamamlandi
      Manuel : Bool;
      AxisReferenced : Bool;   // Servo referansi ayarlandi
   END_VAR
   VAR_OUTPUT
      P1_Ileri : Bool;
      P1_Geri : Bool;
      P2_Ileri : Bool;
      P2_geri : Bool;
      P3_geri : Bool;
      P4_P4B_Geri : Bool;
      ServoGoPos : Bool;
      ClassA_Hazir : Bool;
      ClassE_Hazir : Bool;
      ClassF_Hazir : Bool;
   END_VAR
   VAR_TEMP
      bClassA : Bool;
      bClassA_p1_geri : Bool;
      bClassA_p2_geri : Bool;
      bClassA_p3_geri : Bool;
      bClassA_servo_GoPos : Bool;
      bClassE : Bool;
      bClassE_p1_ileri : Bool;
      bClassE_p2_geri : Bool;
      bClassE_p3_geri : Bool;
      bClassE_servo_GoPos : Bool;
      bClassF : Bool;
      bClassF_p1_ileri : Bool;
      bClassF_p2_ileri : Bool;
      bClassF_p3_geri : Bool;
      bClassF_servo_GoPos : Bool;
      rMaxBoy : Real;
      rMinBoy : Real;
      bBoyOk : Bool;   // Servo Secilen model boy mesafesinde
   END_VAR
BEGIN

REGION Network 1 (SCL)
   #rMaxBoy := "Receipt".CurrentModel.Boy_C + 4;
   #rMinBoy := "Receipt".CurrentModel.Boy_C - 4;

   #bBoyOk := "System_Data".CmdDrive.ActPosition < #rMaxBoy
               AND "System_Data".CmdDrive.ActPosition > #rMinBoy;
END_REGION

REGION Network 2: A modeli
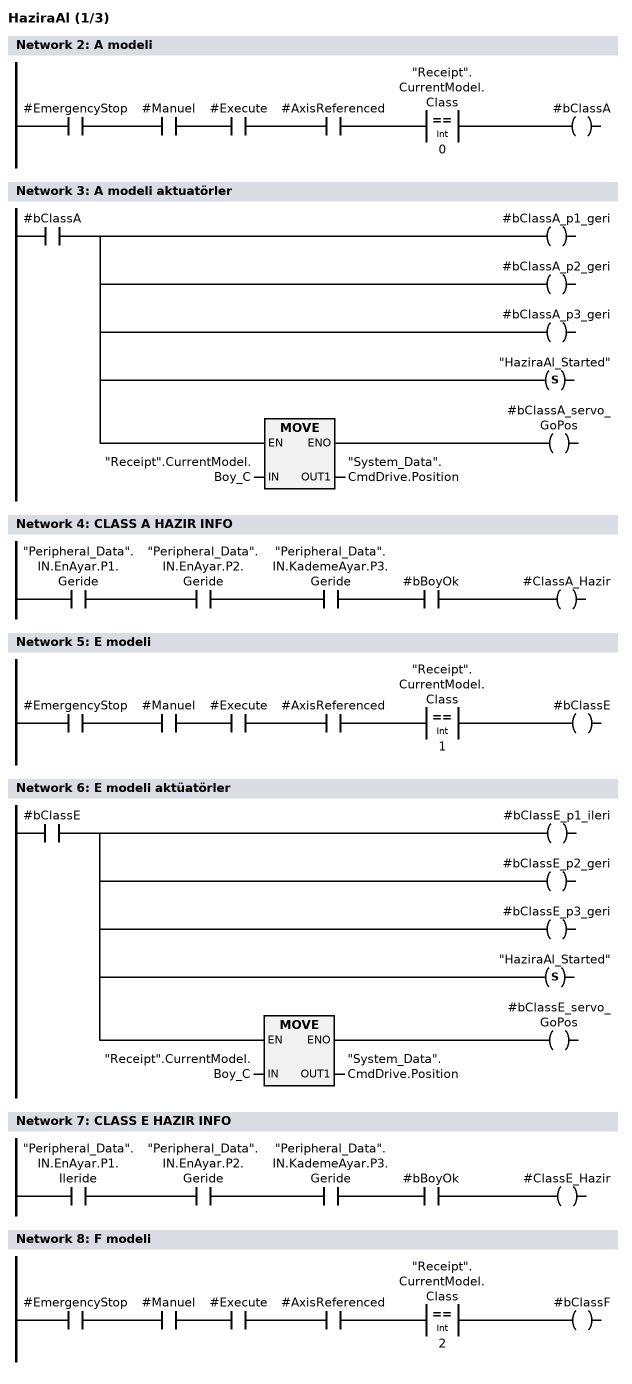
   RUNG wire#powerrail
      Contact( #EmergencyStop )
      Contact( #Manuel )
      Contact( #Execute )
      Contact( #AxisReferenced )
      { S7_Templates := "SrcType := Int" } EQ_Contact(in1 := "Receipt".CurrentModel.Class, in2 := 0)
      Coil( #bClassA )
   END_RUNG
   // the same network as SCL:
   #bClassA := #EmergencyStop AND #Manuel AND #Execute AND #AxisReferenced AND ("Receipt".CurrentModel.Class = 0);
END_REGION

REGION Network 3: A modeli aktuatörler
   RUNG wire#powerrail
      Contact( #bClassA )
      wire#w1
      Coil( #bClassA_p1_geri )
   END_RUNG
   RUNG wire#w1
      Coil( #bClassA_p2_geri )
   END_RUNG
   RUNG wire#w1
      Coil( #bClassA_p3_geri )
   END_RUNG
   RUNG wire#w1
      S_Coil( "HaziraAl_Started" )
   END_RUNG
   RUNG wire#w1
      Move(in := "Receipt".CurrentModel.Boy_C, out1 => "System_Data".CmdDrive.Position)
      Coil( #bClassA_servo_GoPos )
   END_RUNG
   // the same network as SCL:
   #bClassA_p1_geri := #bClassA;
   #bClassA_p2_geri := #bClassA;
   #bClassA_p3_geri := #bClassA;
   IF #bClassA THEN
       "HaziraAl_Started" := TRUE;
       "System_Data".CmdDrive.Position := "Receipt".CurrentModel.Boy_C;
   END_IF;
   #bClassA_servo_GoPos := #bClassA;
END_REGION

REGION Network 4: CLASS A HAZIR INFO
   RUNG wire#powerrail
      Contact( "Peripheral_Data".IN.EnAyar.P1.Geride )
      Contact( "Peripheral_Data".IN.EnAyar.P2.Geride )
      Contact( "Peripheral_Data".IN.KademeAyar.P3.Geride )
      Contact( #bBoyOk )
      Coil( #ClassA_Hazir )
   END_RUNG
   // the same network as SCL:
   #ClassA_Hazir := "Peripheral_Data".IN.EnAyar.P1.Geride AND "Peripheral_Data".IN.EnAyar.P2.Geride AND "Peripheral_Data".IN.KademeAyar.P3.Geride AND #bBoyOk;
END_REGION

REGION Network 5: E modeli
   RUNG wire#powerrail
      Contact( #EmergencyStop )
      Contact( #Manuel )
      Contact( #Execute )
      Contact( #AxisReferenced )
      { S7_Templates := "SrcType := Int" } EQ_Contact(in1 := "Receipt".CurrentModel.Class, in2 := 1)
      Coil( #bClassE )
   END_RUNG
   // the same network as SCL:
   #bClassE := #EmergencyStop AND #Manuel AND #Execute AND #AxisReferenced AND ("Receipt".CurrentModel.Class = 1);
END_REGION

REGION Network 6: E modeli aktüatörler
   RUNG wire#powerrail
      Contact( #bClassE )
      wire#w1
      Coil( #bClassE_p1_ileri )
   END_RUNG
   RUNG wire#w1
      Coil( #bClassE_p2_geri )
   END_RUNG
   RUNG wire#w1
      Coil( #bClassE_p3_geri )
   END_RUNG
   RUNG wire#w1
      S_Coil( "HaziraAl_Started" )
   END_RUNG
   RUNG wire#w1
      Move(in := "Receipt".CurrentModel.Boy_C, out1 => "System_Data".CmdDrive.Position)
      Coil( #bClassE_servo_GoPos )
   END_RUNG
   // the same network as SCL:
   #bClassE_p1_ileri := #bClassE;
   #bClassE_p2_geri := #bClassE;
   #bClassE_p3_geri := #bClassE;
   IF #bClassE THEN
       "HaziraAl_Started" := TRUE;
       "System_Data".CmdDrive.Position := "Receipt".CurrentModel.Boy_C;
   END_IF;
   #bClassE_servo_GoPos := #bClassE;
END_REGION

REGION Network 7: CLASS E HAZIR INFO
   RUNG wire#powerrail
      Contact( "Peripheral_Data".IN.EnAyar.P1.Ileride )
      Contact( "Peripheral_Data".IN.EnAyar.P2.Geride )
      Contact( "Peripheral_Data".IN.KademeAyar.P3.Geride )
      Contact( #bBoyOk )
      Coil( #ClassE_Hazir )
   END_RUNG
   // the same network as SCL:
   #ClassE_Hazir := "Peripheral_Data".IN.EnAyar.P1.Ileride AND "Peripheral_Data".IN.EnAyar.P2.Geride AND "Peripheral_Data".IN.KademeAyar.P3.Geride AND #bBoyOk;
END_REGION

REGION Network 8: F modeli
   RUNG wire#powerrail
      Contact( #EmergencyStop )
      Contact( #Manuel )
      Contact( #Execute )
      Contact( #AxisReferenced )
      { S7_Templates := "SrcType := Int" } EQ_Contact(in1 := "Receipt".CurrentModel.Class, in2 := 2)
      Coil( #bClassF )
   END_RUNG
   // the same network as SCL:
   #bClassF := #EmergencyStop AND #Manuel AND #Execute AND #AxisReferenced AND ("Receipt".CurrentModel.Class = 2);
END_REGION

REGION Network 9: F modeli aktüatörler
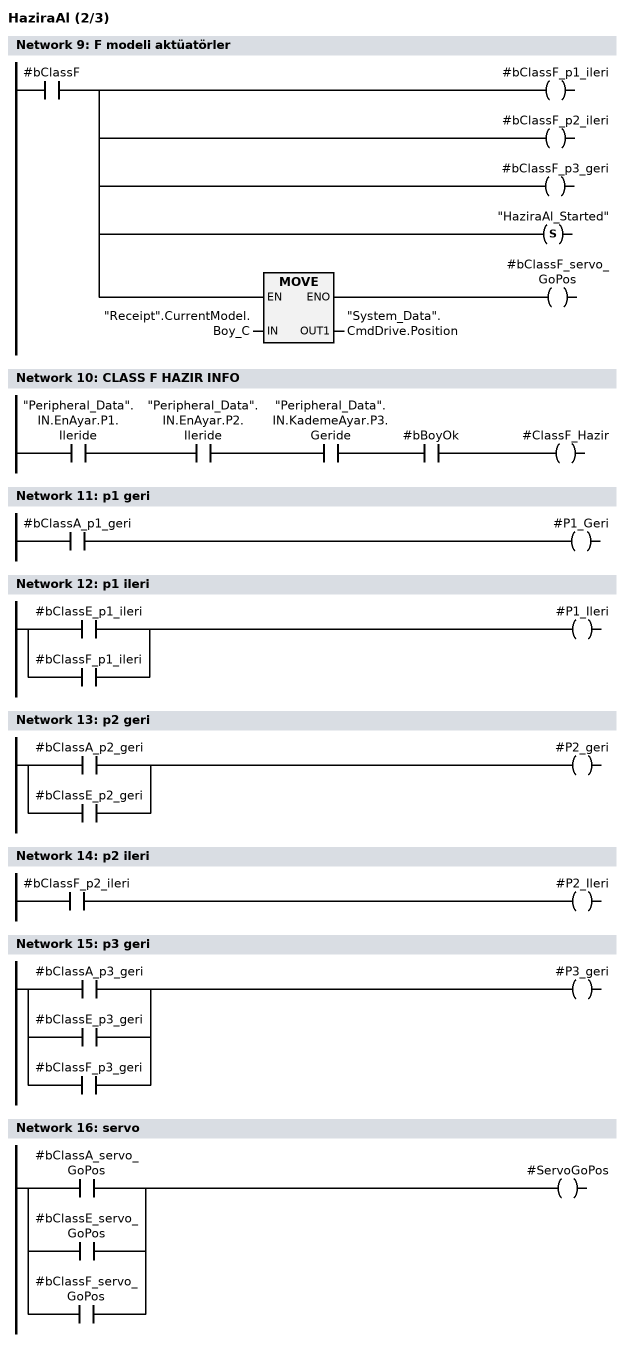
   RUNG wire#powerrail
      Contact( #bClassF )
      wire#w1
      Coil( #bClassF_p1_ileri )
   END_RUNG
   RUNG wire#w1
      Coil( #bClassF_p2_ileri )
   END_RUNG
   RUNG wire#w1
      Coil( #bClassF_p3_geri )
   END_RUNG
   RUNG wire#w1
      S_Coil( "HaziraAl_Started" )
   END_RUNG
   RUNG wire#w1
      Move(in := "Receipt".CurrentModel.Boy_C, out1 => "System_Data".CmdDrive.Position)
      Coil( #bClassF_servo_GoPos )
   END_RUNG
   // the same network as SCL:
   #bClassF_p1_ileri := #bClassF;
   #bClassF_p2_ileri := #bClassF;
   #bClassF_p3_geri := #bClassF;
   IF #bClassF THEN
       "HaziraAl_Started" := TRUE;
       "System_Data".CmdDrive.Position := "Receipt".CurrentModel.Boy_C;
   END_IF;
   #bClassF_servo_GoPos := #bClassF;
END_REGION

REGION Network 10: CLASS F HAZIR INFO
   RUNG wire#powerrail
      Contact( "Peripheral_Data".IN.EnAyar.P1.Ileride )
      Contact( "Peripheral_Data".IN.EnAyar.P2.Ileride )
      Contact( "Peripheral_Data".IN.KademeAyar.P3.Geride )
      Contact( #bBoyOk )
      Coil( #ClassF_Hazir )
   END_RUNG
   // the same network as SCL:
   #ClassF_Hazir := "Peripheral_Data".IN.EnAyar.P1.Ileride AND "Peripheral_Data".IN.EnAyar.P2.Ileride AND "Peripheral_Data".IN.KademeAyar.P3.Geride AND #bBoyOk;
END_REGION

REGION Network 11: p1 geri
   RUNG wire#powerrail
      Contact( #bClassA_p1_geri )
      Coil( #P1_Geri )
   END_RUNG
   // the same network as SCL:
   #P1_Geri := #bClassA_p1_geri;
END_REGION

REGION Network 12: p1 ileri
   RUNG wire#powerrail
      Contact( #bClassE_p1_ileri )
      wire#w1
      Coil( #P1_Ileri )
   END_RUNG
   RUNG wire#powerrail
      Contact( #bClassF_p1_ileri )
   END_RUNG wire#w1
   // the same network as SCL:
   #P1_Ileri := #bClassE_p1_ileri OR #bClassF_p1_ileri;
END_REGION

REGION Network 13: p2 geri
   RUNG wire#powerrail
      Contact( #bClassA_p2_geri )
      wire#w1
      Coil( #P2_geri )
   END_RUNG
   RUNG wire#powerrail
      Contact( #bClassE_p2_geri )
   END_RUNG wire#w1
   // the same network as SCL:
   #P2_geri := #bClassA_p2_geri OR #bClassE_p2_geri;
END_REGION

REGION Network 14: p2 ileri
   RUNG wire#powerrail
      Contact( #bClassF_p2_ileri )
      Coil( #P2_Ileri )
   END_RUNG
   // the same network as SCL:
   #P2_Ileri := #bClassF_p2_ileri;
END_REGION

REGION Network 15: p3 geri
   RUNG wire#powerrail
      Contact( #bClassA_p3_geri )
      wire#w1
      Coil( #P3_geri )
   END_RUNG
   RUNG wire#powerrail
      Contact( #bClassE_p3_geri )
   END_RUNG wire#w1
   RUNG wire#powerrail
      Contact( #bClassF_p3_geri )
   END_RUNG wire#w1
   // the same network as SCL:
   #P3_geri := #bClassA_p3_geri OR #bClassE_p3_geri OR #bClassF_p3_geri;
END_REGION

REGION Network 16: servo
   RUNG wire#powerrail
      Contact( #bClassA_servo_GoPos )
      wire#w1
      Coil( #ServoGoPos )
   END_RUNG
   RUNG wire#powerrail
      Contact( #bClassE_servo_GoPos )
   END_RUNG wire#w1
   RUNG wire#powerrail
      Contact( #bClassF_servo_GoPos )
   END_RUNG wire#w1
   // the same network as SCL:
   #ServoGoPos := #bClassA_servo_GoPos OR #bClassE_servo_GoPos OR #bClassF_servo_GoPos;
END_REGION

REGION Network 17: p4/p4b geri hareket
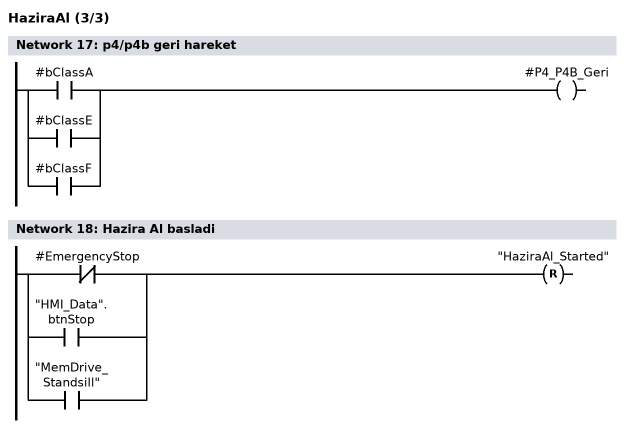
   RUNG wire#powerrail
      Contact( #bClassA )
      wire#w1
      Coil( #P4_P4B_Geri )
   END_RUNG
   RUNG wire#powerrail
      Contact( #bClassE )
   END_RUNG wire#w1
   RUNG wire#powerrail
      Contact( #bClassF )
   END_RUNG wire#w1
   // the same network as SCL:
   #P4_P4B_Geri := #bClassA OR #bClassE OR #bClassF;
END_REGION

REGION Network 18: Hazira Al basladi
   RUNG wire#powerrail
      I_Contact( #EmergencyStop )
      wire#w1
      R_Coil( "HaziraAl_Started" )
   END_RUNG
   RUNG wire#powerrail
      Contact( "HMI_Data".btnStop )
   END_RUNG wire#w1
   RUNG wire#powerrail
      Contact( "MemDrive_Standsill" )
   END_RUNG wire#w1
   // the same network as SCL:
   IF NOT #EmergencyStop OR "HMI_Data".btnStop OR "MemDrive_Standsill" THEN
       "HaziraAl_Started" := FALSE;
   END_IF;
END_REGION
END_FUNCTION

// folder: Receipt

FUNCTION "ReceiptManager" : Void   // FC1, LAD
{ S7_Optimized_Access := 'TRUE' }
VERSION : 0.1
BEGIN

REGION Network 1: Kaydedildi mesaji icin
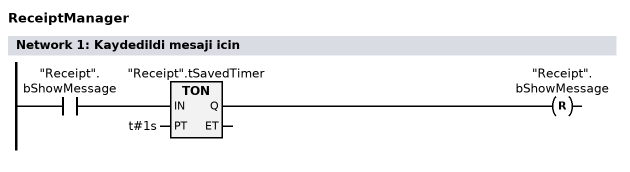
   "Receipt".tSavedTimer.TON(IN := "Receipt".bShowMessage, PT := t#1s);
   IF "Receipt".tSavedTimer.Q THEN "Receipt".bShowMessage := FALSE; END_IF;
END_REGION

REGION Network 2 (SCL): Reçete kontrolu

   // save butonuna basılması
   IF "Receipt".btnSave THEN
       "Receipt".ModelList["Receipt".ModelId].Name := "Receipt".CurrentModel.Name;
       "Receipt".ModelList["Receipt".ModelId].Class := "Receipt".CurrentModel.Class;
       "Receipt".ModelList["Receipt".ModelId].Boy_C := "Receipt".CurrentModel.Boy_C;
       "Receipt".ModelList["Receipt".ModelId].En_D := "Receipt".CurrentModel.En_D;

       "Receipt".btnSave := false;
       "Receipt".bShowMessage := true;
   END_IF;

   // combobox tan model degisimi
   IF "Receipt".OldModelId <> "Receipt".ModelId THEN
       "Receipt".CurrentModel.Name := "Receipt".ModelList["Receipt".ModelId].Name;
       "Receipt".CurrentModel.Class := "Receipt".ModelList["Receipt".ModelId].Class;
       "Receipt".CurrentModel.Boy_C := "Receipt".ModelList["Receipt".ModelId].Boy_C;
       "Receipt".CurrentModel.En_D := "Receipt".ModelList["Receipt".ModelId].En_D;
       "Receipt".OldModelId := "Receipt".ModelId;

       "Receipt".btnSave := false;
       "Receipt".bShowMessage := false;
   END_IF;
END_REGION
END_FUNCTION

(* ===== HMI "HMI_RT_1" =====
system functions are stored by id; their names below are inferred from use
connection "HMI_Connection_2": ETHERNET, SMART_S7_1200_OMS

HMI tags "Default tag table"
   "Tag_ScreenNumber" : UInt, internal
   "ManEnAyarPisIleri" : Bool = PLC ManP1_EnAyar_Ileri AT %M4.0, 1 s
   "btnStartForHmi" : Bool = PLC btnStartForHmi AT %M5.7, 1 s

HMI tags "HmiTags"
   "ModelId" : Int = PLC Receipt.ModelId AT %DB1.DBW0, 500 ms
   "ModelName" : String[50] = PLC Receipt.CurrentModel.Name AT %DB1.DBX0.0, 500 ms
   "Receipt_btnSave" : Bool = PLC Receipt.btnSave, 100 ms
   "Receipt_bShowMessage" : Bool = PLC Receipt.bShowMessage, 100 ms
   "Receipt_CurrentModel_Boy_C" : Real = PLC Receipt.CurrentModel.Boy_C, 100 ms
   "Receipt_CurrentModel_Class" : Int = PLC Receipt.CurrentModel.Class, 100 ms
   "Receipt_CurrentModel_En_D" : Real = PLC Receipt.CurrentModel.En_D, 100 ms
   "HMI_Data_btnAuto" : Bool = PLC HMI_Data.btnAuto, 100 ms
   "HMI_Data_btnManuel" : Bool = PLC HMI_Data.btnManuel, 100 ms
   "HMI_Data_ServoButton_btnGoPos" : Bool = PLC HMI_Data.ServoButton.btnGoPos, 100 ms
   "HMI_Data_ServoButton_btnHataReset" : Bool = PLC HMI_Data.ServoButton.btnHataReset, 100 ms
   "HMI_Data_ServoButton_btnHome" : Bool = PLC HMI_Data.ServoButton.btnHome, 100 ms
   "HMI_Data_ServoButton_btnJogGeri" : Bool = PLC HMI_Data.ServoButton.btnJogGeri, 100 ms
   "HMI_Data_ServoButton_btnJogIleri" : Bool = PLC HMI_Data.ServoButton.btnJogIleri, 100 ms
   "HMI_Data_ServoButton_btnRefNokBelirle" : Bool = PLC HMI_Data.ServoButton.btnRefNokBelirle, 100 ms
   "HMI_Data_ServoData_txtJogOverride" : Int = PLC HMI_Data.ServoData.txtJogOverride, 500 ms
   "HMI_Data_ServoData_txtPozisyon" : Real = PLC HMI_Data.ServoData.txtActPozisyon, 500 ms
   "HMI_Data_ServoData_txtVelocity" : Real = PLC HMI_Data.ServoData.txtVelocity, 500 ms
   "System_Data_CmdDrive_Message" : String[40] = PLC System_Data.CmdDrive.Message, 100 ms
   "HMI_Data.Buttons.btnVakumJeneratoru" : Bool = PLC HMI_Data.Buttons.btnVakumJeneratoru, 100 ms
   "HMI_Data_btnHaziraAl" : Bool = PLC HMI_Data.btnHaziraAl, 100 ms
   "HMI_Data_btnStart" : Bool = PLC HMI_Data.btnStart, 100 ms
   "HMI_Data_btnStop" : Bool = PLC HMI_Data.btnStop, 100 ms
   "HMI_Data_btnVincLambasi" : Bool = PLC HMI_Data.btnVincLambasi, 100 ms
   "HMI_Data_Kademe Pistonu_btnGeri" : Bool = PLC HMI_Data."Kademe Pistonu".btnGeri, 100 ms
   "HMI_Data_Kademe Pistonu_btnIleri" : Bool = PLC HMI_Data."Kademe Pistonu".btnIleri, 100 ms
   "HMI_Data.KenetlemePistonu.P4.btnGeri" : Bool = PLC HMI_Data.KenetlemePistonu.P4.btnGeri, 100 ms
   "HMI_Data.KenetlemePistonu.P4.btnIleri" : Bool = PLC HMI_Data.KenetlemePistonu.P4.btnIleri, 100 ms
   "HMI_Data_KenetlemeSuresi" : Time = PLC HMI_Data.KenetlemeSuresi, 1 s
   "HMI_Data_Status_KademePis_Geride" : Bool = PLC HMI_Data.Status.KademePis_P3.Geride, 1 s
   "HMI_Data_Status_KademePis_Ileride" : Bool = PLC HMI_Data.Status.KademePis_P3.Ileride, 1 s
   "HMI_Data_Status_KenetlemePis_Geride" : Bool = PLC HMI_Data.Status.KenetlemePis_P4.Geride, 1 s
   "HMI_Data_Status_KenetlemePis_Ileride" : Bool = PLC HMI_Data.Status.KenetlemePis_P4.Ileride, 1 s
   "HMI_Data_AcilSayfasi" : Bool = PLC HMI_Data.AcilSayfasi, 100 ms
   "HMI_Data_EnAyarPistonu_P1_btnGeri" : Bool = PLC HMI_Data.EnAyarPistonu.P1.btnGeri, 100 ms
   "HMI_Data_EnAyarPistonu_P1_btnIleri" : Bool = PLC HMI_Data.EnAyarPistonu.P1.btnIleri, 100 ms
   "HMI_Data_EnAyarPistonu_P2_btnGeri" : Bool = PLC HMI_Data.EnAyarPistonu.P2.btnGeri, 100 ms
   "HMI_Data_EnAyarPistonu_P2_btnIleri" : Bool = PLC HMI_Data.EnAyarPistonu.P2.btnIleri, 100 ms
   "HMI_Data_ServoButton_btnKenetle" : Bool = PLC HMI_Data.ServoButton.btnKenetle, 100 ms
   "HMI_Data_ServoButton_btnStop" : Bool = PLC HMI_Data.ServoButton.btnStop, 100 ms
   "HMI_Data_ServoData_txtGerdirmeMes" : Real = PLC HMI_Data.ServoData.txtGerdirmeMes, 500 ms
   "HMI_Data_Status_EnAyarPis_P1_Geride" : Bool = PLC HMI_Data.Status.EnAyarPis.P1.Geride, 1 s
   "HMI_Data_Status_EnAyarPis_P1_Ileride" : Bool = PLC HMI_Data.Status.EnAyarPis.P1.Ileride, 1 s
   "HMI_Data_Status_EnAyarPis_P2_Geride" : Bool = PLC HMI_Data.Status.EnAyarPis.P2.Geride, 1 s
   "HMI_Data_Status_EnAyarPis_P2_Ileride" : Bool = PLC HMI_Data.Status.EnAyarPis.P2.Ileride, 1 s
   "HMI_Data.KenetlemePistonu.P4B.btnGeri" : Bool = PLC HMI_Data.KenetlemePistonu.P4B.btnGeri AT %DB1.DBX0.0, 100 ms
   "HMI_Data.KenetlemePistonu.P4B.btnIleri" : Bool = PLC HMI_Data.KenetlemePistonu.P4B.btnIleri AT %DB1.DBX0.0, 100 ms

HMI tags "System"
   "System_Data_SystemMode_Auto" : Bool = PLC System_Data.SystemMode.Auto, 100 ms
   "System_Data_SystemMode_Man" : Bool = PLC System_Data.SystemMode.Man AT %DB1.DBX0.0, 100 ms
   "System_Data_AutoSeq_Message" : String[50] = PLC System_Data.AutoSeq_Message, 1 s
   "System_Data_CmdDrive_Alarm" : Word = PLC System_Data.CmdDrive.Alarm, 1 s
   "System_Data_CmdDrive_AxisError" : Bool = PLC System_Data.CmdDrive.AxisError, 1 s
   "System_Data_CmdDrive_Error" : Bool = PLC System_Data.CmdDrive.Error, 1 s
   "System_Data_CmdDrive_ReferencedAxis" : Bool = PLC System_Data.CmdDrive.ReferencedAxis, 1 s
   "System_Data_Ready" : Bool = PLC System_Data.Ready, 1 s

HMI tags "Alarms"
   "ServoOrCylinderAlarms" : Word = PLC Alarm_DB.wAlarmsServoOrCylinder AT %DB1.DBW0, 1 s
   "PeripAlarms" : Word = PLC Alarm_DB.wAlarmsPeripheral AT %DB1.DBW0, 1 s

HMI tags "Peripheral"
   "Peripheral_Data.IN.Acil_Stop" : Bool = PLC Peripheral_Data.IN.Acil_Stop AT %DB1.DBW0, 100 ms
   "Peripheral_Data_IN_Acil_Stop" : Bool = PLC Peripheral_Data.IN.Acil_Stop, 100 ms
   "Peripheral_Data_IN_EnAyar_P1_Geride" : Bool = PLC Peripheral_Data.IN.EnAyar.P1.Geride, 1 s
   "Peripheral_Data_IN_EnAyar_P1_Ileride" : Bool = PLC Peripheral_Data.IN.EnAyar.P1.Ileride, 1 s
   "Peripheral_Data_IN_EnAyar_P1A_Geride" : Bool = PLC Peripheral_Data.IN.EnAyar.P1A.Geride, 1 s
   "Peripheral_Data_IN_EnAyar_P1A_Ileride" : Bool = PLC Peripheral_Data.IN.EnAyar.P1A.Ileride, 1 s
   "Peripheral_Data_IN_EnAyar_P2_Geride" : Bool = PLC Peripheral_Data.IN.EnAyar.P2.Geride, 1 s
   "Peripheral_Data_IN_EnAyar_P2_Ileride" : Bool = PLC Peripheral_Data.IN.EnAyar.P2.Ileride, 1 s
   "Peripheral_Data_IN_EnAyar_P2A_Geride" : Bool = PLC Peripheral_Data.IN.EnAyar.P2A.Geride, 1 s
   "Peripheral_Data_IN_EnAyar_P2A_Ileride" : Bool = PLC Peripheral_Data.IN.EnAyar.P2A.Ileride, 1 s
   "Peripheral_Data_IN_KademeAyar_P3_Geride" : Bool = PLC Peripheral_Data.IN.KademeAyar.P3.Geride, 1 s
   "Peripheral_Data_IN_KademeAyar_P3_Ileride" : Bool = PLC Peripheral_Data.IN.KademeAyar.P3.Ileride, 1 s
   "Peripheral_Data_IN_Kenetleme_P4_Geride" : Bool = PLC Peripheral_Data.IN.Kenetleme.P4.Geride, 1 s
   "Peripheral_Data_IN_Kenetleme_P4_Ilderide" : Bool = PLC Peripheral_Data.IN.Kenetleme.P4.Ilderide, 1 s
   "Peripheral_Data_IN_Kenetleme_P4B_Geride" : Bool = PLC Peripheral_Data.IN.Kenetleme.P4B.Geride, 1 s
   "Peripheral_Data_IN_Kenetleme_P4B_Ilderide" : Bool = PLC Peripheral_Data.IN.Kenetleme.P4B.Ilderide, 1 s
   "Peripheral_Data_OUT_LAMBA_Kirmizi" : Bool = PLC Peripheral_Data.OUT.LAMBA.Kirmizi, 1 s
   "Peripheral_Data_OUT_LAMBA_Yesil" : Bool = PLC Peripheral_Data.OUT.LAMBA.Yesil, 1 s
   "Peripheral_Data_OUT_VacumJeneratoru" : Bool = PLC Peripheral_Data.OUT.Vacum, 1 s
   "Peripheral_Data_OUT_VincLambasi" : Bool = PLC Peripheral_Data.OUT.VincLambasi, 1 s
   "Peripheral_Data.OUT.LAMBA.Buzzer" : Bool = PLC Peripheral_Data.OUT.LAMBA.Buzzer, 500 ms
   "Peripheral_Data.OUT.LAMBA.Sari" : Bool = PLC Peripheral_Data.OUT.LAMBA.Sari, 500 ms

discrete alarms
   1: 'P1 pistonu ileri hareket hatasi', class Errors, trigger "ServoOrCylinderAlarms" bit 0
   2: 'P1 pistonu geri hareket hatasi', class Errors, trigger "ServoOrCylinderAlarms" bit 1
   3: 'P2 pistonu ileri hareket hatasi', class Errors, trigger "ServoOrCylinderAlarms" bit 2
   4: 'P2 pistonu geri hareket hatasi', class Errors, trigger "ServoOrCylinderAlarms" bit 3
   5: 'P3 pistonu ileri hareket hatasi', class Errors, trigger "ServoOrCylinderAlarms" bit 4
   6: 'P3 pistonu geri hareket hatasi', class Errors, trigger "ServoOrCylinderAlarms" bit 5
   7: 'P4-P4A pistonu ileri hareket hatasi', class Errors, trigger "ServoOrCylinderAlarms" bit 6
   8: 'P4-P4A pistonu geri hareket hatasi', class Errors, trigger "ServoOrCylinderAlarms" bit 7
   9: 'P4B-P4C pistonu ileri hareket hatasi', class Errors, trigger "ServoOrCylinderAlarms" bit 8
   10: 'P4B-P4C pistonu geri hareket hatasi', class Errors, trigger "ServoOrCylinderAlarms" bit 9
   11: 'Servo sürücü hatasi', class Errors, trigger "ServoOrCylinderAlarms" bit 10
   12: 'ACİL STOP basılı !!! (I0.0)', class Errors, trigger "PeripAlarms" bit 0

text list "textListReceipt": 0 'C100'; 1 'C150'; 2 'C200E'; 3 'C200F'; 4 'C300E'; 5 'C300F'; 6 'C400E'; 7 'C400F'; 8 'C500F'; 9 'C600F'; 10 'REÇETE 1'; 11 'REÇETE 2'; 12 'REÇETE 3'; 13 'REÇETE 4'; 14 'REÇETE 5'; 15 'REÇETE 6'; 16 'REÇETE 7'; 17 'REÇETE 8'; 18 'REÇETE 9'; 19 'REÇETE 10'; 20 'REÇETE 11'

text list "classList": 0 'Boş'; 1 'E'; 2 'F'

Template "MainTemplate" 800x480
   Button "Start screen" at 4,422 size 125x51; TextOff 'Ana Ekran'; TextOn 'Start screen'; PictureOn "NavigateHome_KTP900_Basic_PN_TR"; PictureOff "Home"
      on Click: ActivateScreen("01_Root screen", 0)
   Button "Start screen_1" at 137,422 size 125x51; TextOff 'I/O izleme'; TextOn 'Start screen'; PictureOff "Home"; PictureOn "NavigateHome_KTP900_Basic_PN_TR"
      on Click: ActivateScreen("04_Izleme", 0)
   Button "Start screen_2" at 270,422 size 125x51; TextOff 'Servo Kont.'; TextOn 'Start screen'; PictureOn "NavigateHome_KTP900_Basic_PN_TR"; PictureOff "Home"
      on Click: ActivateScreen("03_Servo", 0)
   Button "Start screen_3" at 404,422 size 125x51; TextOff 'Manuel'; TextOn 'Start screen'; PictureOff "Home"; PictureOn "NavigateHome_KTP900_Basic_PN_TR"
      on Click: ActivateScreen("02_Manuel", 0)
   Button "Start screen_4" at 537,422 size 125x51; TextOff 'Reçete'; TextOn 'Start screen'; PictureOn "NavigateHome_KTP900_Basic_PN_TR"; PictureOff "Home"
      on Click: ActivateScreen("05_Receipt", 0)
   Button "Start screen_5" at 671,422 size 125x51; TextOff 'Alarm'; TextOn 'Start screen'; PictureOff "Home"; PictureOn "NavigateHome_KTP900_Basic_PN_TR"
      on Click: ActivateScreen("06_Alarm", 0)

screen "01_Root screen" 800x480, template "MainTemplate"
   on GenerateScreen: SetTag("Tag_ScreenNumber", 1)
   Rectangle "Template_Rectangle_1" at 0,0 size 800x480
      Visibility <- "HMI_Data_AcilSayfasi"
   TextField "Text field_5" at 282,262 size 233x34; Text 'ACİL STOP BASILI'
      Visibility <- "HMI_Data_AcilSayfasi"
   GraphicView "Graphic view_1" at 335,129 size 137x121; Picture "warning"
      Visibility <- "HMI_Data_AcilSayfasi"
   TextField "Template_Text field_4" at 45,139 size 175x23; Text 'Servo Anlık Pozisyon'
   Group "Group_2" at 0,132 size 799x37
   Button "Button_1" at 17,266 size 222x57; TextOff 'MANUEL'
      on Press: function_b14e0dd5("HMI_Data_btnManuel", 0)
      Appearance <- "System_Data_SystemMode_Man"
   Button "Button_3" at 289,266 size 222x57; TextOff 'STOP'
      on Press: function_b14e0dd5("HMI_Data_btnStop", 0)
   Button "Button_4" at 558,267 size 222x55; TextOff 'HAZIRA AL'
      on Press: function_b14e0dd5("HMI_Data_btnHaziraAl", 0)
      Appearance <- "System_Data_Ready"
   Button "Button_5" at 17,341 size 222x57; TextOff 'OTOMATİK'
      Appearance <- "System_Data_SystemMode_Auto"
      on Press: function_b14e0dd5("HMI_Data_btnAuto", 0)
   TextField "Text field_1" at 55,234 size 146x20; Text 'ÇALIŞMA MODU'
   TextField "Text field_2" at 320,234 size 164x20; Text 'SİSTEM STOP'
   TextField "Text field_3" at 595,235 size 146x20; Text 'EK SİSTEM'
   TextField "Text field_4" at 46,62 size 135x23; Text 'Sistem Durumu:'
   IOField "I/O field_1" at 270,59 size 525x32; FormatPattern ??????????????????????????????????????????????????
      ProcessValue <- "System_Data_AutoSeq_Message"
   TextField "Template_Text field_1" at 45,102 size 123x23; Text 'Seçilen Model:'
   DateTimeField "HmiScreenItemData" at 656,26 size 139x20
   DateTimeField "HmiScreenItemData_1" at 657,2 size 133x20
   GraphicView "Template_Graphic view_1" at 5,5 size 122x48; Picture "isikoglu_logo4"
   TextField "Template_Text field_2" at 265,9 size 312x34; Text 'KENETLEME MAKİNESİ 1'
   IOField "I/O field_2" at 270,97 size 525x32; FormatPattern ??????????????????????????????????????????????????
      ProcessValue <- "ModelName"
   Button "Button_2" at 289,340 size 222x55; TextOff 'START'
      on Press: function_b14e0dd5("btnStartForHmi", 0)
   IOField "I/O field_3" at 417,133 size 253x37; FormatPattern 999999999.99; Unit  mm
      ProcessValue <- "HMI_Data_ServoData_txtPozisyon"

screen "02_Manuel" 800x480, template "MainTemplate"
   TextField "Text field_1" at 25,3 size 221x20; Text 'En Ayar Pistonu Kademe 1 (P1)'
   Button "Button_3" at 26,91 size 214x55; TextOff 'Geri'
      on Press: function_b14e0dd5("HMI_Data_EnAyarPistonu_P1_btnGeri", 0)
   Button "Button_1" at 26,28 size 214x55; TextOff 'İleri'
      on Press: function_b14e0dd5("HMI_Data_EnAyarPistonu_P1_btnIleri", 0)
   Rectangle "Rectangle_2" at 242,28 size 13x55
      Appearance <- "HMI_Data_Status_EnAyarPis_P1_Ileride"
   Rectangle "Rectangle_3" at 242,91 size 13x55
      Appearance <- "HMI_Data_Status_EnAyarPis_P1_Geride"
   Button "Button_2" at 290,91 size 214x55; TextOff 'Geri'
      on Press: function_b14e0dd5("HMI_Data.KenetlemePistonu.P4.btnGeri", 0)
   Button "Button_4" at 290,28 size 214x55; TextOff 'İleri'
      on Press: function_b14e0dd5("HMI_Data.KenetlemePistonu.P4.btnIleri", 0)
   Rectangle "Rectangle_5" at 506,28 size 13x55
      Appearance <- "Peripheral_Data_IN_Kenetleme_P4_Ilderide"
   Rectangle "Rectangle_6" at 506,91 size 13x55
      Appearance <- "Peripheral_Data_IN_Kenetleme_P4_Geride"
   TextField "Text field_13" at 288,3 size 225x20; Text 'Kenetleme Pistonu (P4) (SAĞ)'
   Button "Button_5" at 553,92 size 214x55; TextOff 'Geri'
      on Press: function_b14e0dd5("HMI_Data_Kademe Pistonu_btnGeri", 0)
   Button "Button_6" at 553,29 size 214x55; TextOff 'İleri'
      on Press: function_b14e0dd5("HMI_Data_Kademe Pistonu_btnIleri", 0)
   Rectangle "Rectangle_8" at 769,29 size 13x55
      Appearance <- "HMI_Data_Status_KademePis_Ileride"
   Rectangle "Rectangle_9" at 769,92 size 13x55
      Appearance <- "HMI_Data_Status_KademePis_Geride"
   TextField "Text field_8" at 586,3 size 146x20; Text 'Kademe Pistonu (P3)'
   TextField "Text field_2" at 81,161 size 108x20; Text 'Vinç Lambası'
   Button "Button_8" at 26,186 size 214x55; TextOff 'Aktif / Pasif'
      on Release: InvertBit("HMI_Data_btnVincLambasi")
   Rectangle "Rectangle_11" at 244,186 size 11x55
      Appearance <- "Peripheral_Data_OUT_VincLambasi"
   Button "Button_7" at 290,186 size 214x55; TextOff 'Aktif / Pasif'
      on Release: InvertBit("HMI_Data.Buttons.btnVakumJeneratoru")
   Rectangle "Rectangle_17" at 506,186 size 13x55
      Appearance <- "Peripheral_Data_OUT_VacumJeneratoru"
   TextField "Text field_3" at 331,162 size 140x20; Text 'Vakum Jeneratoru'
   TextField "Text field_5" at 27,257 size 222x20; Text 'En Ayar Pistonu Kademe 2 (P2)'
   Button "Button_9" at 26,345 size 214x55; TextOff 'Geri'
      on Press: function_b14e0dd5("HMI_Data_EnAyarPistonu_P2_btnGeri", 0)
   Button "Button_10" at 26,282 size 214x55; TextOff 'İleri'
      on Press: function_b14e0dd5("HMI_Data_EnAyarPistonu_P2_btnIleri", 0)
   Rectangle "Rectangle_18" at 242,282 size 13x55
      Appearance <- "HMI_Data_Status_EnAyarPis_P2_Ileride"
   Rectangle "Rectangle_19" at 242,345 size 13x55
      Appearance <- "HMI_Data_Status_EnAyarPis_P2_Geride"
   Button "Button_11" at 290,345 size 214x55; TextOff 'Geri'
      on Press: function_b14e0dd5("HMI_Data.KenetlemePistonu.P4B.btnGeri", 0)
   Button "Button_12" at 290,282 size 214x55; TextOff 'İleri'
      on Press: function_b14e0dd5("HMI_Data.KenetlemePistonu.P4B.btnIleri", 0)
   Rectangle "Rectangle_20" at 506,282 size 13x55
      Appearance <- "Peripheral_Data_IN_Kenetleme_P4B_Ilderide"
   Rectangle "Rectangle_21" at 506,345 size 13x55
      Appearance <- "Peripheral_Data_IN_Kenetleme_P4B_Geride"
   TextField "Text field_6" at 288,257 size 227x20; Text 'Kenetleme Pistonu (P4B) (SOL)'
   Rectangle "Template_Rectangle_2" at 0,0 size 800x480
      Visibility <- "HMI_Data_AcilSayfasi"
   TextField "Text field_4" at 282,262 size 233x34; Text 'ACİL STOP BASILI'
      Visibility <- "HMI_Data_AcilSayfasi"
   GraphicView "Graphic view_1" at 335,129 size 137x121; Picture "kisspng-icon-danger-tape-cliparts-5a7c86e0694cb3.3733218515181104324313"
      Visibility <- "HMI_Data_AcilSayfasi"

screen "03_Servo" 800x480, template "MainTemplate"
   Button "Button_1" at 131,80 size 132x77; TextOff 'JOG Geri'
      on Press: function_b14e0dd5("HMI_Data_ServoButton_btnJogGeri", 0)
   IOField "I/O field_1" at 346,118 size 104x39; FormatPattern 999; Unit  %
      ProcessValue <- "HMI_Data_ServoData_txtJogOverride"
   IOField "I/O field_2" at 273,80 size 253x37; FormatPattern 999999999.99
      ProcessValue <- "HMI_Data_ServoData_txtPozisyon"
   Button "Button_5" at 534,80 size 132x77; TextOff 'JOG İleri'
      on Press: function_b14e0dd5("HMI_Data_ServoButton_btnJogIleri", 0)
   Button "btnIncJogSpeedXaxis" at 269,119 size 74x37; TextOff '-'
      on Release: function_b9b71300("HMI_Data_ServoData_txtJogOverride", 5)
   Button "Button_3" at 453,119 size 75x37; TextOff '+'
      on Release: function_dd21b452("HMI_Data_ServoData_txtJogOverride", 5)
   Button "Button_4" at 173,223 size 150x71; TextOff 'HOME GİT'
      on Press: function_b14e0dd5("HMI_Data_ServoButton_btnHome", 0)
   Button "Button_8" at 17,223 size 150x71; TextOff 'REFERANS NOKTASI BELİRLE'
      on Press: function_b14e0dd5("HMI_Data_ServoButton_btnRefNokBelirle", 0)
      Appearance <- "System_Data_CmdDrive_ReferencedAxis"
   Button "Button_9" at 329,223 size 150x71; TextOff 'MODEL POZİSYONUNA GİT'
      on Press: function_b14e0dd5("HMI_Data_ServoButton_btnGoPos", 0)
   Button "Button_13" at 640,223 size 150x71; TextOff 'HATA RESET'
      on Press: function_b14e0dd5("HMI_Data_ServoButton_btnHataReset", 0)
      Appearance <- "System_Data_CmdDrive_AxisError"
   TextField "Text field_1" at 295,46 size 227x20; Text 'SERVO MANUEL KONTROL'
   TextField "Text field_2" at 299,180 size 227x20; Text 'SERVO KOMUTLARI'
   TextField "Text field_5" at 295,46 size 227x20; Text 'SERVO MANUEL KONTROL'
   Button "Button_6" at 484,223 size 150x71; TextOff 'KENETLEME POZİSYONUNA GİT'
      on Press: function_b14e0dd5("HMI_Data_ServoButton_btnKenetle", 0)
   Button "Button_2" at 292,325 size 222x57; TextOff 'STOP'
      on Press: function_b14e0dd5("HMI_Data_ServoButton_btnStop", 0)
   TextField "Text field_3" at 12,10 size 111x22; Text 'Servo Durumu'
   IOField "I/O field_3" at 147,4 size 633x32; FormatPattern ????????????????????????????????????????
      ProcessValue <- "System_Data_CmdDrive_Message"
   Rectangle "Template_Rectangle_2" at 0,0 size 800x480
      Visibility <- "HMI_Data_AcilSayfasi"
   TextField "Text field_7" at 282,262 size 233x34; Text 'ACİL STOP BASILI'
      Visibility <- "HMI_Data_AcilSayfasi"
   GraphicView "Graphic view_1" at 335,129 size 137x121; Picture "kisspng-icon-danger-tape-cliparts-5a7c86e0694cb3.3733218515181104324313"
      Visibility <- "HMI_Data_AcilSayfasi"

screen "04_Izleme" 800x480, template "MainTemplate"
   TextField "Text field_1" at 81,3 size 108x20; Text 'En Ayar Pistonu'
   TextField "Text field_2" at 139,27 size 51x20; Text 'İleride'
   Circle "Circle_1" at 148,52 size 34x34
      Appearance <- "Peripheral_Data_IN_EnAyar_P1_Ileride"
   TextField "Text field_3" at 200,27 size 51x20; Text 'Geride'
   Circle "Circle_2" at 209,52 size 34x34
      Appearance <- "Peripheral_Data_IN_EnAyar_P1_Geride"
   Circle "Circle_3" at 148,96 size 34x34
      Appearance <- "Peripheral_Data_IN_EnAyar_P2_Ileride"
   Circle "Circle_4" at 209,96 size 34x34
      Appearance <- "Peripheral_Data_IN_EnAyar_P2_Geride"
   TextField "Text field_4" at 42,60 size 60x20; Text 'P1 (sol):'
   TextField "Text field_5" at 43,101 size 65x20; Text 'P2 (sağ):'
   Circle "Circle_5" at 148,138 size 34x34
      Appearance <- "Peripheral_Data_IN_EnAyar_P1A_Ileride"
   Circle "Circle_6" at 209,138 size 34x34
      Appearance <- "Peripheral_Data_IN_EnAyar_P1A_Geride"
   Circle "Circle_7" at 148,182 size 34x34
      Appearance <- "Peripheral_Data_IN_EnAyar_P2A_Ileride"
   Circle "Circle_8" at 209,182 size 34x34
      Appearance <- "Peripheral_Data_IN_EnAyar_P2A_Geride"
   TextField "Text field_6" at 42,146 size 70x20; Text 'P1A (sol):'
   TextField "Text field_7" at 43,187 size 75x20; Text 'P2A (sağ):'
   TextField "Text field_8" at 606,3 size 108x20; Text 'Kademe Pistonu'
   TextField "Text field_9" at 664,27 size 51x20; Text 'İleride'
   Circle "Circle_9" at 673,52 size 34x34
      Appearance <- "Peripheral_Data_IN_KademeAyar_P3_Ileride"
   TextField "Text field_10" at 725,27 size 51x20; Text 'Geride'
   Circle "Circle_10" at 734,52 size 34x34
      Appearance <- "Peripheral_Data_IN_KademeAyar_P3_Geride"
   TextField "Text field_11" at 567,60 size 26x20; Text 'P3:'
   TextField "Text field_13" at 318,2 size 155x20; Text 'Kenetleme Pistonu'
   TextField "Text field_14" at 401,26 size 51x20; Text 'İleride'
   Circle "Circle_13" at 410,51 size 34x34
      Appearance <- "Peripheral_Data_IN_Kenetleme_P4_Ilderide"
   TextField "Text field_15" at 462,26 size 51x20; Text 'Geride'
   Circle "Circle_14" at 471,51 size 34x34
      Appearance <- "Peripheral_Data_IN_Kenetleme_P4_Geride"
   TextField "Text field_16" at 304,59 size 65x20; Text 'P4 (sağ):'
   Circle "Circle_17" at 410,96 size 34x34
      Appearance <- "Peripheral_Data_IN_Kenetleme_P4B_Ilderide"
   Circle "Circle_18" at 471,96 size 34x34
      Appearance <- "Peripheral_Data_IN_Kenetleme_P4B_Geride"
   TextField "Text field_18" at 304,104 size 68x20; Text 'P4B (sol):'
   TextField "Text field_20" at 81,231 size 108x20; Text 'İkaz Lambaları'
   Circle "Circle_21" at 178,260 size 34x34
      Appearance <- "Peripheral_Data_OUT_LAMBA_Yesil"
   TextField "Text field_23" at 42,268 size 40x20; Text 'Yeşil:'
   TextField "Text field_21" at 322,231 size 155x20; Text 'Diğer Ekipmanlar'
   Circle "Circle_22" at 441,261 size 34x34
      Appearance <- "Peripheral_Data_OUT_VacumJeneratoru"
   TextField "Text field_22" at 304,268 size 53x20; Text 'Vakum:'
   Circle "Circle_24" at 441,305 size 34x34
      Appearance <- "Peripheral_Data_OUT_VincLambasi"
   TextField "Text field_25" at 304,311 size 93x20; Text 'Vinc Lambası:'
   Circle "Circle_25" at 177,305 size 34x34
      Appearance <- "Peripheral_Data.OUT.LAMBA.Sari"
   TextField "Text field_26" at 42,310 size 35x20; Text 'Sarı:'
   Circle "Circle_11" at 440,351 size 34x34
      Appearance <- "Peripheral_Data.OUT.LAMBA.Buzzer"
   TextField "Text field_12" at 305,356 size 43x20; Text 'Siren:'
   Circle "Circle_23" at 178,351 size 34x34
      Appearance <- "Peripheral_Data_OUT_LAMBA_Kirmizi"
   TextField "Text field_24" at 43,356 size 51x20; Text 'Kırmızı:'

